(* IEC 61131-3 sources: RL_MAR/experiments/results/ablation/Ablation_random_topo_deepseek-ai_DeepSeek-V3.2_20260603_051006, 94 files *)

(* ---- hard_92.st ---- *)
FUNCTION_BLOCK FB_BreakerControlSystem
VAR_INPUT
    B10_1_Trip : BOOL;
    B10_1_Close : BOOL;
    B10_2_Trip : BOOL;
    B10_2_Close : BOOL;
    B10_12_Trip : BOOL;
    B10_12_Close : BOOL;
    B54_Trip : BOOL;
    B54_Close : BOOL;
    B55_Trip : BOOL;
    B55_Close : BOOL;
    B56_Trip : BOOL;
    B56_Close : BOOL;
    B57_Trip : BOOL;
    B57_Close : BOOL;
END_VAR

VAR_OUTPUT
    Point_1a : INT;
    Point_2a : INT;
    Point_3a : INT;
    Point_4a : INT;
    B10_1_Opened : BOOL;
    B10_1_Closed : BOOL;
    B10_2_Opened : BOOL;
    B10_2_Closed : BOOL;
    B10_12_Opened : BOOL;
    B10_12_Closed : BOOL;
    B54_Opened : BOOL;
    B54_Closed : BOOL;
    B55_Opened : BOOL;
    B55_Closed : BOOL;
    B56_Opened : BOOL;
    B56_Closed : BOOL;
    B57_Opened : BOOL;
    B57_Closed : BOOL;
END_VAR

VAR
    SEL86_OUT : INT;
    MOVE89_OUT : INT;
    SEL66_OUT : INT;
    MOVE69_OUT : INT;
    SEL96_OUT : INT;
    MOVE99_OUT : INT;
    SEL106_OUT : INT;
    MOVE109_OUT : INT;
END_VAR

// Breaker state transitions
IF B10_1_Close THEN
    B10_1_Closed := TRUE;
    B10_1_Opened := FALSE;
ELSIF B10_1_Trip THEN
    B10_1_Closed := FALSE;
    B10_1_Opened := TRUE;
END_IF;

IF B10_2_Close THEN
    B10_2_Closed := TRUE;
    B10_2_Opened := FALSE;
ELSIF B10_2_Trip THEN
    B10_2_Closed := FALSE;
    B10_2_Opened := TRUE;
END_IF;

IF B10_12_Close THEN
    B10_12_Closed := TRUE;
    B10_12_Opened := FALSE;
ELSIF B10_12_Trip THEN
    B10_12_Closed := FALSE;
    B10_12_Opened := TRUE;
END_IF;

IF B54_Close THEN
    B54_Closed := TRUE;
    B54_Opened := FALSE;
ELSIF B54_Trip THEN
    B54_Closed := FALSE;
    B54_Opened := TRUE;
END_IF;

IF B55_Close THEN
    B55_Closed := TRUE;
    B55_Opened := FALSE;
ELSIF B55_Trip THEN
    B55_Closed := FALSE;
    B55_Opened := TRUE;
END_IF;

IF B56_Close THEN
    B56_Closed := TRUE;
    B56_Opened := FALSE;
ELSIF B56_Trip THEN
    B56_Closed := FALSE;
    B56_Opened := TRUE;
END_IF;

IF B57_Close THEN
    B57_Closed := TRUE;
    B57_Opened := FALSE;
ELSIF B57_Trip THEN
    B57_Closed := FALSE;
    B57_Opened := TRUE;
END_IF;

// Point calculations
// Point_1a: B54 closed AND (B10_12 closed AND B10_1 closed) OR B10_2 closed
IF B54_Closed AND ((B10_12_Closed AND B10_1_Closed) OR B10_2_Closed) THEN
    Point_1a := 0;
ELSE
    Point_1a := 138;
END_IF;

// Point_2a: B55 closed AND (B10_12 closed AND B10_1 closed) OR B10_2 closed
IF B55_Closed AND ((B10_12_Closed AND B10_1_Closed) OR B10_2_Closed) THEN
    Point_2a := 0;
ELSE
    Point_2a := 138;
END_IF;

// Point_3a: B56 closed AND (B10_12 closed AND B10_2 closed) OR B10_1 closed
IF B56_Closed AND ((B10_12_Closed AND B10_2_Closed) OR B10_1_Closed) THEN
    Point_3a := 0;
ELSE
    Point_3a := 138;
END_IF;

// Point_4a: B57 closed AND (B10_12 closed AND B10_2 closed) OR B10_1 closed
IF B57_Closed AND ((B10_12_Closed AND B10_2_Closed) OR B10_1_Closed) THEN
    Point_4a := 0;
ELSE
    Point_4a := 138;
END_IF;

END_FUNCTION_BLOCK

(* ---- hard_93.st ---- *)
FUNCTION_BLOCK FB_CircuitControl
VAR_INPUT
    Reset_All_CB : BOOL;
    Current_Fault_on_TRSF1 : INT;
    Current_Fault_on_66BUS1 : INT;
END_VAR

VAR_OUTPUT
    Short_Circuit_TRSF1 : BOOL;
    Short_Circuit_66BUS : BOOL;
    Open_CB1_66KV : BOOL;
    Open_CB2_66KV : BOOL;
    Open_CB_TRSF1 : BOOL;
    Open_CB2_22KV : BOOL;
END_VAR

VAR
    Threshold500 : INT := 500;
    Prev_Open_CB2_22KV : BOOL;
    Prev_Open_CB1_66KV : BOOL;
    Prev_Open_CB_TRSF1 : BOOL;
    Temp_Open_CB2_22KV : BOOL;
    Temp_Open_CB1_66KV : BOOL;
    Temp_Open_CB_TRSF1 : BOOL;
END_VAR

(* a) Implement short circuit detection *)
Short_Circuit_66BUS := (Current_Fault_on_66BUS1 > Threshold500);
Short_Circuit_TRSF1 := (Current_Fault_on_TRSF1 > Threshold500);

(* b) Implement circuit breaker control logic *)

(* First pass: Initial calculations *)
Temp_Open_CB2_22KV := (NOT Reset_All_CB) AND (NOT Prev_Open_CB2_22KV) AND (
    (Open_CB1_66KV AND Open_CB_TRSF1) OR Short_Circuit_66BUS
);

Temp_Open_CB1_66KV := (NOT Reset_All_CB) AND (NOT Temp_Open_CB2_22KV) AND (
    (Prev_Open_CB1_66KV AND Open_CB_TRSF1) OR Short_Circuit_66BUS
);

Temp_Open_CB_TRSF1 := (NOT Reset_All_CB) AND (NOT Temp_Open_CB2_22KV) AND (
    (Temp_Open_CB1_66KV AND Prev_Open_CB_TRSF1) OR Short_Circuit_66BUS
);

Open_CB2_66KV := TRUE;

(* Second pass: Update based on new conditions *)
Temp_Open_CB2_22KV := Temp_Open_CB2_22KV OR (
    (NOT Reset_All_CB) AND (NOT Prev_Open_CB2_22KV) AND (
        (Open_CB2_66KV AND Temp_Open_CB1_66KV AND Temp_Open_CB_TRSF1) OR Short_Circuit_TRSF1
    )
);

Temp_Open_CB1_66KV := Temp_Open_CB1_66KV OR (
    (NOT Reset_All_CB) AND (NOT Temp_Open_CB2_22KV) AND (
        (Open_CB2_66KV AND Prev_Open_CB1_66KV AND Temp_Open_CB_TRSF1) OR Short_Circuit_TRSF1
    )
);

Temp_Open_CB_TRSF1 := Temp_Open_CB_TRSF1 OR (
    (NOT Reset_All_CB) AND (NOT Temp_Open_CB2_22KV) AND (
        (Open_CB2_66KV AND Temp_Open_CB1_66KV AND Prev_Open_CB_TRSF1) OR Short_Circuit_TRSF1
    )
);

(* Assign temporary values to outputs *)
Open_CB2_22KV := Temp_Open_CB2_22KV;
Open_CB1_66KV := Temp_Open_CB1_66KV;
Open_CB_TRSF1 := Temp_Open_CB_TRSF1;

(* Store previous states for next scan *)
Prev_Open_CB2_22KV := Open_CB2_22KV;
Prev_Open_CB1_66KV := Open_CB1_66KV;
Prev_Open_CB_TRSF1 := Open_CB_TRSF1;

(* Failsafe: If Reset_All_CB is TRUE, force all circuit breakers to FALSE *)
IF Reset_All_CB THEN
    Open_CB1_66KV := FALSE;
    Open_CB2_66KV := FALSE;
    Open_CB_TRSF1 := FALSE;
    Open_CB2_22KV := FALSE;
    Prev_Open_CB2_22KV := FALSE;
    Prev_Open_CB1_66KV := FALSE;
    Prev_Open_CB_TRSF1 := FALSE;
END_IF;

END_FUNCTION_BLOCK

(* ---- hard_94.st ---- *)
FUNCTION_BLOCK FB_AdvancedCircuitBreakerControl
VAR_INPUT
    S_AL1_P_B1 : BOOL;
    S_AL1_P_B2 : BOOL;
    S_AL1_MCB : BOOL;
    MCB_BUSY : BOOL;
    MCB_ERROR : BOOL;
    S_AL1_MCBR : BOOL;
    MCBR_BUSY : BOOL;
    MCBR_ERROR : BOOL;
    S_AL1_P_B3 : BOOL;
    S_AL1_MCB2 : BOOL;
    S_AL1_MCBR2 : BOOL;
END_VAR

VAR_OUTPUT
    E_AL1_B1 : BOOL;
    PUWS_AL1_B1_PLUS : BOOL;
    PUWS_AL1_B1_RIGHT : BOOL;
    PAS_AL1_PLUS : BOOL;
    PAS_AL1_TURN : BOOL;
END_VAR

VAR
    PPAL1 : BOOL := 1;
    PP0 : BOOL := 1;
    PP1 : BOOL := 0;
    PP2 : BOOL := 0;
    PP3 : BOOL := 0;
    PP4 : BOOL := 0;
    MCB : BOOL := 1;
    PP5 : BOOL := 0;
    PP7 : BOOL := 0;
    PPL3 : BOOL := 0;
    PPL4 : BOOL := 0;
    MCBR : BOOL := 1;
    PPL5 : BOOL := 0;
    PPL7 : BOOL := 0;
    STABLE : BOOL := 0;
    MCB_CONTROL : BOOL;
END_VAR

STABLE := 0;
WHILE (STABLE = 0) DO
    STABLE := 1;

    IF (PP0 = 1) AND (NOT MCB_CONTROL) AND (NOT PP1) THEN
        PP0 := 0;
        PP1 := 1;
        STABLE := 0;
    END_IF;

    IF (PP1 = 1) AND S_AL1_P_B1 AND (NOT PP2) THEN
        PP1 := 0;
        PP2 := 1;
        STABLE := 0;
    END_IF;

    IF (PP2 = 1) AND S_AL1_P_B2 AND (NOT MCB_CONTROL) AND (NOT PP3) THEN
        PP2 := 0;
        PP3 := 1;
        STABLE := 0;
    END_IF;

    IF (PP2 = 1) AND S_AL1_P_B2 AND MCB_CONTROL AND (NOT PPL3) AND (NOT PP1) THEN
        PP2 := 0;
        PPL3 := 1;
        PP1 := 1;
        STABLE := 0;
    END_IF;

    IF (PP3 = 1) AND S_AL1_MCB AND (NOT PP4) AND (NOT PP1) THEN
        PP3 := 0;
        PP4 := 1;
        PP1 := 1;
        STABLE := 0;
    END_IF;

    IF (PP4 = 1) AND (MCB = 1) AND MCB_BUSY AND (NOT PP5) THEN
        PP4 := 0;
        MCB := 0;
        PP5 := 1;
        STABLE := 0;
    END_IF;

    IF (PP5 = 1) AND S_AL1_MCB2 AND (NOT PP7) AND (NOT MCB) THEN
        PP5 := 0;
        PP7 := 1;
        MCB := 1;
        STABLE := 0;
    END_IF;

    IF (PP7 = 1) AND S_AL1_P_B3 THEN
        PP7 := 0;
        STABLE := 0;
    END_IF;

    IF (PPL3 = 1) AND S_AL1_MCBR AND (NOT PPL4) THEN
        PPL3 := 0;
        PPL4 := 1;
        STABLE := 0;
    END_IF;

    IF (PPL4 = 1) AND (MCBR = 1) AND MCBR_BUSY AND (NOT PPL5) THEN
        PPL4 := 0;
        MCBR := 0;
        PPL5 := 1;
        STABLE := 0;
    END_IF;

    IF (PPL5 = 1) AND S_AL1_MCBR2 AND (NOT PPL7) AND (NOT MCBR) THEN
        PPL5 := 0;
        PPL7 := 1;
        MCBR := 1;
        STABLE := 0;
    END_IF;

    IF (PPL7 = 1) AND S_AL1_P_B3 THEN
        PPL7 := 0;
        STABLE := 0;
    END_IF;
END_WHILE;

IF (PP0 = 1) OR (PP1 = 1) THEN
    E_AL1_B1 := 1;
END_IF;

IF (PP3 = 1) THEN
    MCB_CONTROL := 1;
END_IF;

IF (PPL3 = 1) OR (PPL4 = 1) THEN
    PAS_AL1_PLUS := 1;
    PAS_AL1_TURN := 1;
END_IF;

IF (PPAL1 = 1) OR (PP2 = 1) THEN
    PUWS_AL1_B1_PLUS := 1;
END_IF;

IF (PP2 = 1) OR (PP3 = 1) OR (PPL3 = 1) THEN
    E_AL1_B1 := 0;
END_IF;

IF (PP0 = 1) OR (PP3 = 1) THEN
    MCB_CONTROL := 0;
END_IF;

IF (PP0 = 1) OR (PP3 = 1) OR (PP4 = 1) THEN
    PAS_AL1_PLUS := 0;
    PAS_AL1_TURN := 0;
END_IF;

IF (PPAL1 = 1) OR (PP2 = 1) THEN
    PUWS_AL1_B1_RIGHT := 0;
END_IF;

END_FUNCTION_BLOCK

(* ---- hf_1.st ---- *)
FUNCTION_BLOCK StackMin
VAR_INPUT
    push : BOOL;
    pop : BOOL;
    reset : BOOL;
END_VAR
VAR_OUTPUT
    error : BOOL;
    status : WORD;
END_VAR
VAR_IN_OUT
    item : INT;
    stack : ARRAY[0..3] OF INT;
END_VAR
VAR
    top : INT := -1;
    i : INT;
    minIndex : INT;
    minValue : INT;
    j : INT;
END_VAR

// Reset operation takes highest priority
IF reset THEN
    top := -1;
    error := FALSE;
    status := 16#0000;
ELSIF push THEN
    // Push operation
    IF top >= 3 THEN
        // Stack is full
        error := TRUE;
        status := 16#8A04;
    ELSE
        // Add item to stack
        top := top + 1;
        stack[top] := item;
        error := FALSE;
        status := 16#0000;
    END_IF;
ELSIF pop THEN
    // Pop minimum operation
    IF top < 0 THEN
        // Stack is empty
        error := TRUE;
        status := 16#8A05;
    ELSE
        // Find minimum value and its index
        minIndex := 0;
        minValue := stack[0];

        FOR i := 1 TO top DO
            IF stack[i] < minValue THEN
                minValue := stack[i];
                minIndex := i;
            END_IF;
        END_FOR;

        // Return minimum value via item
        item := minValue;

        // Shift elements down to remove the minimum
        FOR j := minIndex TO top - 1 DO
            stack[j] := stack[j + 1];
        END_FOR;

        // Clear the last position (optional but clean)
        stack[top] := 0;

        // Update top index
        top := top - 1;

        error := FALSE;
        status := 16#0000;
    END_IF;
ELSE
    // No operation requested
    error := FALSE;
    status := 16#0000;
END_IF;
END_FUNCTION_BLOCK

(* ---- hf_10.st ---- *)
FUNCTION_BLOCK FloatingAverage
VAR_INPUT
    cyclicExecution : BOOL;
    trigger : BOOL;
    value : REAL;
    windowSize : INT;
    reset : BOOL;
END_VAR
VAR_OUTPUT
    average : REAL;
    windowSizeReached : BOOL;
    error : BOOL;
    status : WORD;
END_VAR
VAR
    dataBuffer : ARRAY[1..100] OF REAL;
    bufferIndex : INT;
    sum : REAL;
    elementCount : INT;
    prevTrigger : BOOL;
END_VAR

// Initialize variables
bufferIndex := 1;
sum := 0.0;
elementCount := 0;
prevTrigger := FALSE;
average := 0.0;
windowSizeReached := FALSE;
error := FALSE;
status := 16#0000;

// Check for reset condition
IF reset THEN
    bufferIndex := 1;
    sum := 0.0;
    elementCount := 0;
    average := 0.0;
    windowSizeReached := FALSE;
    error := FALSE;
    status := 16#0000;
    RETURN;
END_IF;

// Validate window size
IF (windowSize < 1) OR (windowSize > 100) THEN
    error := TRUE;
    status := 16#8200;
    average := 0.0;
    windowSizeReached := FALSE;
    RETURN;
END_IF;

// Check if we should process new data
IF cyclicExecution OR (trigger AND NOT prevTrigger) THEN
    // Store previous value that will be overwritten
    IF elementCount >= windowSize THEN
        sum := sum - dataBuffer[bufferIndex];
    END_IF;

    // Store new value and update sum
    dataBuffer[bufferIndex] := value;
    sum := sum + value;

    // Update element count
    IF elementCount < windowSize THEN
        elementCount := elementCount + 1;
    END_IF;

    // Update buffer index (circular buffer)
    bufferIndex := bufferIndex + 1;
    IF bufferIndex > windowSize THEN
        bufferIndex := 1;
    END_IF;

    // Calculate average
    IF elementCount > 0 THEN
        average := sum / elementCount;
    ELSE
        average := 0.0;
    END_IF;

    // Check if window size is reached
    windowSizeReached := (elementCount >= windowSize);
END_IF;

// Store current trigger state for edge detection
prevTrigger := trigger;

// Clear error if window size is valid
IF NOT ((windowSize < 1) OR (windowSize > 100)) THEN
    error := FALSE;
    status := 16#0000;
END_IF;

END_FUNCTION_BLOCK

(* ---- hf_11.st ---- *)
FUNCTION_BLOCK FB_BottleProcessing
VAR_INPUT
    bottleSensor : BOOL;
    cleaningConfirmButton : BOOL;
    fillingConfirmButton : BOOL;
    cappingConfirmButton : BOOL;
    packingConfirmButton : BOOL;
    finishedButton : BOOL;
END_VAR

VAR_OUTPUT
    Pump_Motor : BOOL;
    Filling_Valve : BOOL;
    Capping_Machine : BOOL;
    Packing_Machine : BOOL;
    Completion_Light : BOOL;
END_VAR

VAR
    State : INT := 0; (* 0=Waiting, 1=Cleaning, 2=Filling, 3=Capping, 4=Packing, 5=Completed *)
END_VAR

CASE State OF
    0: (* Waiting State *)
        Pump_Motor := FALSE;
        Filling_Valve := FALSE;
        Capping_Machine := FALSE;
        Packing_Machine := FALSE;
        Completion_Light := FALSE;

        IF bottleSensor THEN
            Pump_Motor := TRUE;
            State := 1;
        END_IF;

    1: (* Cleaning State *)
        Pump_Motor := TRUE;
        Filling_Valve := FALSE;
        Capping_Machine := FALSE;
        Packing_Machine := FALSE;
        Completion_Light := FALSE;

        IF cleaningConfirmButton THEN
            Pump_Motor := FALSE;
            Filling_Valve := TRUE;
            State := 2;
        END_IF;

    2: (* Filling State *)
        Pump_Motor := FALSE;
        Filling_Valve := TRUE;
        Capping_Machine := FALSE;
        Packing_Machine := FALSE;
        Completion_Light := FALSE;

        IF fillingConfirmButton THEN
            Filling_Valve := FALSE;
            Capping_Machine := TRUE;
            State := 3;
        END_IF;

    3: (* Capping State *)
        Pump_Motor := FALSE;
        Filling_Valve := FALSE;
        Capping_Machine := TRUE;
        Packing_Machine := FALSE;
        Completion_Light := FALSE;

        IF cappingConfirmButton THEN
            Capping_Machine := FALSE;
            Packing_Machine := TRUE;
            State := 4;
        END_IF;

    4: (* Packing State *)
        Pump_Motor := FALSE;
        Filling_Valve := FALSE;
        Capping_Machine := FALSE;
        Packing_Machine := TRUE;
        Completion_Light := FALSE;

        IF packingConfirmButton THEN
            Packing_Machine := FALSE;
            Completion_Light := TRUE;
            State := 5;
        END_IF;

    5: (* Completed State *)
        Pump_Motor := FALSE;
        Filling_Valve := FALSE;
        Capping_Machine := FALSE;
        Packing_Machine := FALSE;
        Completion_Light := TRUE;

        IF finishedButton THEN
            Completion_Light := FALSE;
            State := 0;
        END_IF;

END_CASE;

END_FUNCTION_BLOCK

(* ---- hf_12.st ---- *)
FUNCTION_BLOCK MaterialMixing
VAR_INPUT
    estop : BOOL; (* Emergency Stop Signal, FALSE: Emergency stop triggered, TRUE: No emergency stop triggered *)
    opeMode : BOOL; (* Operation Mode, FALSE: Manual Operation Mode, TRUE: Automatic Operation Mode *)
    valveAStart : BOOL; (* Valve A Start Button *)
    valveBStart : BOOL; (* Valve B Start Button *)
    valveCStart : BOOL; (* Valve C Start Button *)
    valveDStart : BOOL; (* Valve D Start Button *)
    mixMotorStart : BOOL; (* Mixing Motor Start Button *)
    autoStart : BOOL; (* Automatic Start Button *)
    processMode : BOOL; (* Process Mode *)
    levelSensor : INT; (* Liquid Level Sensor, unit cm *)
    mixMotorComplete : BOOL; (* Mixing Complete Signal *)
END_VAR
VAR_OUTPUT
    valveARun : BOOL; (* Valve A Run Command *)
    valveBRun : BOOL; (* Valve B Run Command *)
    valveCRun : BOOL; (* Valve C Run Command *)
    valveDRun : BOOL; (* Valve D Run Command *)
    mixMotorRun : BOOL; (* Mixing Motor Run Command *)
END_VAR
VAR
    previousValveAStart : BOOL := FALSE;
    previousValveBStart : BOOL := FALSE;
    previousValveCStart : BOOL := FALSE;
    previousValveDStart : BOOL := FALSE;
    previousMixMotorStart : BOOL := FALSE;
    previousAutoStart : BOOL := FALSE;
    autoActive : BOOL := FALSE;
    autoStep : INT := 0;
END_VAR

(* Emergency stop logic - highest priority *)
IF NOT estop THEN
    valveARun := FALSE;
    valveBRun := FALSE;
    valveCRun := FALSE;
    valveDRun := FALSE;
    mixMotorRun := FALSE;
    autoActive := FALSE;
    autoStep := 0;
ELSE
    (* Manual mode *)
    IF NOT opeMode THEN
        (* Valve A toggle control *)
        IF valveAStart AND NOT previousValveAStart THEN
            valveARun := NOT valveARun;
        END_IF;
        previousValveAStart := valveAStart;

        (* Valve B toggle control *)
        IF valveBStart AND NOT previousValveBStart THEN
            valveBRun := NOT valveBRun;
        END_IF;
        previousValveBStart := valveBStart;

        (* Valve C toggle control *)
        IF valveCStart AND NOT previousValveCStart THEN
            valveCRun := NOT valveCRun;
        END_IF;
        previousValveCStart := valveCStart;

        (* Valve D toggle control *)
        IF valveDStart AND NOT previousValveDStart THEN
            valveDRun := NOT valveDRun;
        END_IF;
        previousValveDStart := valveDStart;

        (* Mixing motor toggle control *)
        IF mixMotorStart AND NOT previousMixMotorStart THEN
            mixMotorRun := NOT mixMotorRun;
        END_IF;
        previousMixMotorStart := mixMotorStart;

        (* Reset automatic mode variables in manual mode *)
        autoActive := FALSE;
        autoStep := 0;

    (* Automatic mode *)
    ELSE
        (* Auto start button handling - toggle functionality *)
        IF autoStart AND NOT previousAutoStart THEN
            autoActive := NOT autoActive;
            IF autoActive THEN
                autoStep := 1;
            ELSE
                autoStep := 0;
            END_IF;
        END_IF;
        previousAutoStart := autoStart;

        (* Automatic process sequence *)
        IF autoActive THEN
            CASE autoStep OF
                1: (* Step 1: Open valve A *)
                    valveARun := TRUE;
                    valveBRun := FALSE;
                    valveCRun := FALSE;
                    valveDRun := FALSE;
                    mixMotorRun := FALSE;

                    IF levelSensor >= 50 THEN
                        valveARun := FALSE;
                        autoStep := 2;
                    END_IF;

                2: (* Step 2: Open valve B *)
                    valveBRun := TRUE;

                    IF levelSensor >= 80 THEN
                        valveBRun := FALSE;
                        autoStep := 3;
                    END_IF;

                3: (* Step 3: Process mode decision *)
                    IF NOT processMode THEN
                        (* Process mode false: Start mixing motor *)
                        mixMotorRun := TRUE;

                        IF mixMotorComplete THEN
                            mixMotorRun := FALSE;
                            autoStep := 4;
                        END_IF;
                    ELSE
                        (* Process mode true: Open valve C *)
                        valveCRun := TRUE;

                        IF levelSensor >= 100 THEN
                            valveCRun := FALSE;
                            autoStep := 4;
                        END_IF;
                    END_IF;

                4: (* Step 4: Handle mixing for process mode true *)
                    IF processMode THEN
                        mixMotorRun := TRUE;

                        IF mixMotorComplete THEN
                            mixMotorRun := FALSE;
                            autoStep := 5;
                        END_IF;
                    ELSE
                        autoStep := 5;
                    END_IF;

                5: (* Step 5: Open valve D and end process *)
                    valveDRun := TRUE;
                    autoActive := FALSE;
                    autoStep := 0;

            END_CASE;
        ELSE
            (* Auto not active - ensure all outputs are off *)
            valveARun := FALSE;
            valveBRun := FALSE;
            valveCRun := FALSE;
            valveDRun := FALSE;
            mixMotorRun := FALSE;
        END_IF;
    END_IF;
END_IF;

END_FUNCTION_BLOCK

(* ---- hf_13.st ---- *)
FUNCTION_BLOCK TON
VAR_INPUT
    IN : BOOL;
    PT : DINT;
    CYCLE_TIME : DINT;
END_VAR
VAR_OUTPUT
    Q : BOOL;
    ET : DINT;
END_VAR
VAR
    elapsedTimeInternal : DINT := 0;
    IN_PREV : BOOL := FALSE;
END_VAR

IF IN THEN
    IF NOT IN_PREV THEN
        elapsedTimeInternal := 0;
    END_IF;

    IF elapsedTimeInternal < PT THEN
        elapsedTimeInternal := elapsedTimeInternal + CYCLE_TIME;
        Q := FALSE;
    ELSE
        elapsedTimeInternal := PT;
        Q := TRUE;
    END_IF;

    ET := elapsedTimeInternal;
ELSE
    Q := FALSE;
    ET := 0;
    elapsedTimeInternal := 0;
END_IF;

IN_PREV := IN;
END_FUNCTION_BLOCK

FUNCTION_BLOCK LightsControl
VAR_INPUT
    button1 : BOOL; (* Button 1: Automatic/Manual Mode Select *)
    button2 : BOOL; (* Button 2: Manual Control/Green Light Req *)
    button3 : BOOL; (* Button 3: Manual Control/Red Light Req *)
    CYCLE_TIME : DINT; (* Time elapsed in current cycle (in ms) *)
END_VAR
VAR_OUTPUT
    greenLight : BOOL; (* Green light *)
    redLight : BOOL; (* Red light *)
    yellowLight : BOOL; (* Yellow light *)
END_VAR
VAR
    (* Timers for control *)
    timerAuto : TON;
    timerGreen : TON;
    timerRed : TON;
    timerYellow : TON;

    currentState : INT := 0;
    autoRunTimer : BOOL := TRUE;

    (* Internal variables for blinking control *)
    blinkToggleRed : BOOL := FALSE;
    blinkToggleYellow : BOOL := FALSE;
    blinkToggleGreen : BOOL := FALSE;
    prevTimerRedQ : BOOL := FALSE;
    prevTimerYellowQ : BOOL := FALSE;
    prevTimerGreenQ : BOOL := FALSE;
END_VAR

(* Reset all outputs initially *)
greenLight := FALSE;
redLight := FALSE;
yellowLight := FALSE;

IF button1 THEN (* Automatic Mode *)
    (* Reset manual mode timers *)
    timerGreen(IN := FALSE, PT := 0, CYCLE_TIME := CYCLE_TIME);
    timerRed(IN := FALSE, PT := 0, CYCLE_TIME := CYCLE_TIME);
    timerYellow(IN := FALSE, PT := 0, CYCLE_TIME := CYCLE_TIME);

    (* Reset blinking toggle variables *)
    blinkToggleRed := FALSE;
    blinkToggleYellow := FALSE;
    blinkToggleGreen := FALSE;

    (* Automatic mode state machine *)
    timerAuto(IN := autoRunTimer, PT := 1000, CYCLE_TIME := CYCLE_TIME);

    CASE currentState OF
        0: (* State 0: Green light ON for 1 second *)
            greenLight := TRUE;
            redLight := FALSE;
            yellowLight := FALSE;

            IF timerAuto.Q THEN
                currentState := 1;
                timerAuto(IN := FALSE, PT := 1000, CYCLE_TIME := CYCLE_TIME);
            END_IF;

        1: (* State 1: Red light ON for 1 second *)
            greenLight := FALSE;
            redLight := TRUE;
            yellowLight := FALSE;

            IF timerAuto.Q THEN
                currentState := 2;
                timerAuto(IN := FALSE, PT := 1000, CYCLE_TIME := CYCLE_TIME);
            END_IF;

        2: (* State 2: Yellow light ON for 1 second *)
            greenLight := FALSE;
            redLight := FALSE;
            yellowLight := TRUE;

            IF timerAuto.Q THEN
                currentState := 0;
                timerAuto(IN := FALSE, PT := 1000, CYCLE_TIME := CYCLE_TIME);
            END_IF;
    END_CASE;

    (* Restart timer for next cycle *)
    IF NOT timerAuto.IN THEN
        timerAuto(IN := TRUE, PT := 1000, CYCLE_TIME := CYCLE_TIME);
    END_IF;

ELSE (* Manual Mode *)
    (* Reset automatic mode timer *)
    timerAuto(IN := FALSE, PT := 0, CYCLE_TIME := CYCLE_TIME);

    (* Reset automatic mode state *)
    currentState := 0;

    (* Manual mode logic based on button combinations *)
    IF NOT button2 AND NOT button3 THEN
        (* Both FALSE: All lights off *)
        greenLight := FALSE;
        redLight := FALSE;
        yellowLight := FALSE;

        (* Reset all timers and blinking states *)
        timerGreen(IN := FALSE, PT := 0, CYCLE_TIME := CYCLE_TIME);
        timerRed(IN := FALSE, PT := 0, CYCLE_TIME := CYCLE_TIME);
        timerYellow(IN := FALSE, PT := 0, CYCLE_TIME := CYCLE_TIME);
        blinkToggleRed := FALSE;
        blinkToggleYellow := FALSE;
        blinkToggleGreen := FALSE;

    ELSIF button2 AND NOT button3 THEN
        (* button2 TRUE, button3 FALSE: Green light ON, Red light blinking at 0.5Hz *)
        greenLight := TRUE;
        yellowLight := FALSE;

        (* Red light blinking logic *)
        timerRed(IN := TRUE, PT := 2000, CYCLE_TIME := CYCLE_TIME);

        (* Detect rising edge of timer output to toggle blink *)
        IF timerRed.Q AND NOT prevTimerRedQ THEN
            blinkToggleRed := NOT blinkToggleRed;
        END_IF;
        prevTimerRedQ := timerRed.Q;

        (* Red light blinks at 0.5Hz using timer Q directly *)
        redLight := blinkToggleRed;

        (* Reset other timers *)
        timerGreen(IN := FALSE, PT := 0, CYCLE_TIME := CYCLE_TIME);
        timerYellow(IN := FALSE, PT := 0, CYCLE_TIME := CYCLE_TIME);
        blinkToggleYellow := FALSE;
        blinkToggleGreen := FALSE;

    ELSIF NOT button2 AND button3 THEN
        (* button2 FALSE, button3 TRUE: Red light ON, Yellow light blinking at 1Hz *)
        redLight := TRUE;
        greenLight := FALSE;

        (* Yellow light blinking logic *)
        timerYellow(IN := TRUE, PT := 1000, CYCLE_TIME := CYCLE_TIME);

        (* Detect rising edge of timer output to toggle blink *)
        IF timerYellow.Q AND NOT prevTimerYellowQ THEN
            blinkToggleYellow := NOT blinkToggleYellow;
        END_IF;
        prevTimerYellowQ := timerYellow.Q;

        (* Yellow light blinks at 1Hz using NOT timer Q *)
        yellowLight := blinkToggleYellow;

        (* Reset other timers *)
        timerGreen(IN := FALSE, PT := 0, CYCLE_TIME := CYCLE_TIME);
        timerRed(IN := FALSE, PT := 0, CYCLE_TIME := CYCLE_TIME);
        blinkToggleRed := FALSE;
        blinkToggleGreen := FALSE;

    ELSIF button2 AND button3 THEN
        (* Both TRUE: Yellow light ON, Green light blinking at 1Hz *)
        yellowLight := TRUE;
        redLight := FALSE;

        (* Green light blinking logic *)
        timerGreen(IN := TRUE, PT := 1000, CYCLE_TIME := CYCLE_TIME);

        (* Detect rising edge of timer output to toggle blink *)
        IF timerGreen.Q AND NOT prevTimerGreenQ THEN
            blinkToggleGreen := NOT blinkToggleGreen;
        END_IF;
        prevTimerGreenQ := timerGreen.Q;

        (* Green light blinks at 1Hz using NOT timer Q *)
        greenLight := blinkToggleGreen;

        (* Reset other timers *)
        timerRed(IN := FALSE, PT := 0, CYCLE_TIME := CYCLE_TIME);
        timerYellow(IN := FALSE, PT := 0, CYCLE_TIME := CYCLE_TIME);
        blinkToggleRed := FALSE;
        blinkToggleYellow := FALSE;
    END_IF;
END_IF;
END_FUNCTION_BLOCK

(* ---- hf_14.st ---- *)
FUNCTION_BLOCK TruckGarage
VAR_INPUT
    enter_flag : BOOL;
    exit_flag : BOOL;
    VehicleNumber_in : INT;
END_VAR
VAR_OUTPUT
    truck_row : INT;
    truck_col : INT;
    truck_VehicleNumber : INT;
END_VAR
VAR_IN_OUT
    garage : ARRAY[1..3, 1..5] OF STRUCT
        Occupied : BOOL;
        VehicleNumber : INT;
    END_STRUCT;
END_VAR
VAR
    i : INT;
    j : INT;
    space_found : BOOL;
    exit_found : BOOL;
END_VAR

// Initialize output variables
truck_row := 0;
truck_col := 0;
truck_VehicleNumber := 0;

// Entry logic
IF enter_flag THEN
    space_found := FALSE;

    // Search from last row to first row
    FOR i := 3 TO 1 BY -1 DO
        // Search from last column to first column
        FOR j := 5 TO 1 BY -1 DO
            IF NOT garage[i, j].Occupied THEN
                // Found empty space
                garage[i, j].Occupied := TRUE;
                garage[i, j].VehicleNumber := VehicleNumber_in;
                space_found := TRUE;
                EXIT;
            END_IF;
        END_FOR;

        IF space_found THEN
            EXIT;
        END_IF;
    END_FOR;
END_IF;

// Exit logic
IF exit_flag THEN
    exit_found := FALSE;

    // Search from first row to last row
    FOR i := 1 TO 3 DO
        // Search from first column to last column
        FOR j := 1 TO 5 DO
            IF garage[i, j].Occupied AND garage[i, j].VehicleNumber = VehicleNumber_in THEN
                // Found vehicle to exit
                truck_row := i;
                truck_col := j;
                truck_VehicleNumber := garage[i, j].VehicleNumber;

                // Clear the parking space
                garage[i, j].Occupied := FALSE;
                garage[i, j].VehicleNumber := 0;

                exit_found := TRUE;
                EXIT;
            END_IF;
        END_FOR;

        IF exit_found THEN
            EXIT;
        END_IF;
    END_FOR;
END_IF;
END_FUNCTION_BLOCK

(* ---- hf_15.st ---- *)
FUNCTION_BLOCK FB_MergeBytes
VAR_INPUT
    byteArray : ARRAY[1..20] OF DINT; (* Byte array to be merged *)
END_VAR
VAR_OUTPUT
    dwordArray : ARRAY[1..10] OF DINT; (* Merged double word array *)
    mergeDwordNum : DINT; (* Actual number of merged double words *)
END_VAR
VAR
    i, j, k : DINT; (* Changed from INT to DINT to match array indices *)
    tempDword : DINT;
    currentByteValue : DINT;
END_VAR
VAR CONSTANT
    BYTE_ARRAY_SIZE : DINT := 20; (* Size of the input byte array *)
    DWORD_ARRAY_SIZE : DINT := 10; (* Size of the output DINT array *)
END_VAR

(* Main logic for merging bytes into double words *)
mergeDwordNum := 0;
tempDword := 0;

(* Calculate maximum possible double words from byte array *)
IF BYTE_ARRAY_SIZE >= 4 THEN
    FOR i := 1 TO BYTE_ARRAY_SIZE DO
        (* Extract current byte value (mask to keep only lowest 8 bits) *)
        currentByteValue := byteArray[i] AND 16#FF;

        (* Position byte within double word *)
        CASE (i MOD 4) OF
            1: (* First byte - least significant *)
                tempDword := currentByteValue;

            2: (* Second byte *)
                tempDword := tempDword OR (currentByteValue SHL 8);

            3: (* Third byte *)
                tempDword := tempDword OR (currentByteValue SHL 16);

            0: (* Fourth byte - most significant *)
                tempDword := tempDword OR (currentByteValue SHL 24);

                (* Store completed double word if space available *)
                IF mergeDwordNum < DWORD_ARRAY_SIZE THEN
                    mergeDwordNum := mergeDwordNum + 1;
                    dwordArray[mergeDwordNum] := tempDword;
                END_IF;

                tempDword := 0; (* Reset for next double word *)
        END_CASE;
    END_FOR;
END_IF;

(* Clear remaining positions in dwordArray if any *)
FOR k := (mergeDwordNum + 1) TO DWORD_ARRAY_SIZE DO
    dwordArray[k] := 0;
END_FOR;

END_FUNCTION_BLOCK

(* ---- hf_16.st ---- *)
FUNCTION_BLOCK FB_LinearizeValue
VAR_INPUT
    InputValue : REAL; // Floating point input, raw measurement value
END_VAR

VAR_OUTPUT
    LinearizedValue : REAL; // Converted linear value
    Error : BOOL; // Error status indicator
    Status : WORD; // Status code
END_VAR

VAR
    // Internal constants for readability and maintainability
    InputMin : REAL := 1200.0;
    InputMax : REAL := 7000.0;
    OutputMin : REAL := 150.0;
    OutputMax : REAL := 720.0;

    // Pre-calculated slopes for each segment for efficiency
    Slope1 : REAL := (240.0 - 150.0) / (3600.0 - 1200.0); // 90/2400
    Slope2 : REAL := (560.0 - 240.0) / (4800.0 - 3600.0); // 320/1200
    Slope3 : REAL := (720.0 - 560.0) / (7000.0 - 4800.0); // 160/2200
END_VAR

// Main execution logic
IF InputValue < InputMin THEN
    // Below minimum range
    LinearizedValue := OutputMin;
    Error := TRUE;
    Status := 16#8001;
ELSIF InputValue > InputMax THEN
    // Above maximum range
    LinearizedValue := OutputMax;
    Error := TRUE;
    Status := 16#8001;
ELSE
    // Input is within valid range
    Error := FALSE;
    Status := 16#0000;

    // Determine which segment the input falls into
    IF InputValue <= 3600.0 THEN
        // Range 1: 1200 to 3600
        LinearizedValue := 150.0 + (InputValue - 1200.0) * Slope1;
    ELSIF InputValue <= 4800.0 THEN
        // Range 2: 3600 to 4800
        LinearizedValue := 240.0 + (InputValue - 3600.0) * Slope2;
    ELSE
        // Range 3: 4800 to 7000
        LinearizedValue := 560.0 + (InputValue - 4800.0) * Slope3;
    END_IF;
END_IF;

END_FUNCTION_BLOCK

(* ---- hf_17.st ---- *)
FUNCTION_BLOCK FB_WarehouseManagement
VAR_INPUT
    requestIn : BOOL := FALSE;
    requestOut : BOOL := FALSE;
END_VAR

VAR_OUTPUT
    productNum : INT := 0;
    libFreeNum : INT := 9;
    error : BOOL := FALSE;
    status : WORD := 16#0000;
END_VAR

VAR_IN_OUT
    library : ARRAY[1..9] OF BOOL;
END_VAR

VAR
    i : INT;
    found : BOOL;
    errFull : WORD := 16#8001;
    errEmpty : WORD := 16#8002;
    initDone : BOOL := FALSE;
END_VAR

// Reset error status at start of each cycle
error := FALSE;
status := 16#0000;

// Initialize library array on first execution
IF NOT initDone THEN
    i := 1;
    WHILE i <= 9 DO
        library[i] := FALSE;
        i := i + 1;
    END_WHILE;
    initDone := TRUE;
END_IF;

// Handle product storage request
IF requestIn AND NOT requestOut THEN
    // Check if storage is full
    IF productNum >= 9 THEN
        error := TRUE;
        status := errFull;
    ELSE
        // Search for free position from highest to lowest index (First-In-Last-Out)
        found := FALSE;
        i := 9;
        WHILE i >= 1 AND NOT found DO
            IF NOT library[i] THEN
                library[i] := TRUE;
                productNum := productNum + 1;
                libFreeNum := libFreeNum - 1;
                found := TRUE;
            END_IF;
            i := i - 1;
        END_WHILE;

        // If no free position found (should not happen with proper checks)
        IF NOT found THEN
            error := TRUE;
            status := errFull;
        END_IF;
    END_IF;
END_IF;

// Handle product retrieval request
IF requestOut AND NOT requestIn THEN
    // Check if storage is empty
    IF productNum <= 0 THEN
        error := TRUE;
        status := errEmpty;
    ELSE
        // Search for occupied position from lowest to highest index (First-In-First-Out)
        found := FALSE;
        i := 1;
        WHILE i <= 9 AND NOT found DO
            IF library[i] THEN
                library[i] := FALSE;
                productNum := productNum - 1;
                libFreeNum := libFreeNum + 1;
                found := TRUE;
            END_IF;
            i := i + 1;
        END_WHILE;

        // If no occupied position found (should not happen with proper checks)
        IF NOT found THEN
            error := TRUE;
            status := errEmpty;
        END_IF;
    END_IF;
END_IF;

// Handle concurrent requests (both true) - prioritize storage
IF requestIn AND requestOut THEN
    // Check if storage is full for storage operation
    IF productNum >= 9 THEN
        error := TRUE;
        status := errFull;
    ELSE
        // Perform storage operation (same logic as above)
        found := FALSE;
        i := 9;
        WHILE i >= 1 AND NOT found DO
            IF NOT library[i] THEN
                library[i] := TRUE;
                productNum := productNum + 1;
                libFreeNum := libFreeNum - 1;
                found := TRUE;
            END_IF;
            i := i - 1;
        END_WHILE;

        IF NOT found THEN
            error := TRUE;
            status := errFull;
        END_IF;
    END_IF;
END_IF;

END_FUNCTION_BLOCK

(* ---- hf_18.st ---- *)
FUNCTION_BLOCK FB_ColorLightControl
VAR_INPUT
    controlButton : BOOL; // Push button for sequence control
END_VAR

VAR_OUTPUT
    greenLight : BOOL; // Green light control signal
    redLight : BOOL; // Red light control signal
    yellowLight : BOOL; // Yellow light control signal
END_VAR

VAR
    state : INT := 1; // State machine control variable
    lastControlButton : BOOL := FALSE; // Previous button state for edge detection
END_VAR

// Main logic
IF (controlButton = TRUE) AND (lastControlButton = FALSE) THEN
    // Rising edge detected - execute state transition
    CASE state OF
        1: // State 1: Green Only -> Transition to State 2
            greenLight := FALSE;
            redLight := TRUE;
            yellowLight := FALSE;
            state := 2;

        2: // State 2: Red Only -> Transition to State 3
            greenLight := FALSE;
            redLight := FALSE;
            yellowLight := TRUE;
            state := 3;

        3: // State 3: Yellow Only -> Transition to State 4
            greenLight := TRUE;
            redLight := TRUE;
            yellowLight := TRUE;
            state := 4;

        4: // State 4: All Lights On -> Transition to State 5
            greenLight := FALSE;
            redLight := FALSE;
            yellowLight := FALSE;
            state := 5;

        5: // State 5: All Lights Off -> Transition to State 1
            greenLight := TRUE;
            redLight := FALSE;
            yellowLight := FALSE;
            state := 1;
    END_CASE;
ELSE
    // No rising edge - maintain current state outputs
    CASE state OF
        1: // State 1: Green Only
            greenLight := TRUE;
            redLight := FALSE;
            yellowLight := FALSE;

        2: // State 2: Red Only
            greenLight := FALSE;
            redLight := TRUE;
            yellowLight := FALSE;

        3: // State 3: Yellow Only
            greenLight := FALSE;
            redLight := FALSE;
            yellowLight := TRUE;

        4: // State 4: All Lights On
            greenLight := TRUE;
            redLight := TRUE;
            yellowLight := TRUE;

        5: // State 5: All Lights Off
            greenLight := FALSE;
            redLight := FALSE;
            yellowLight := FALSE;
    END_CASE;
END_IF;

// Update lastControlButton for next cycle's edge detection
lastControlButton := controlButton;

END_FUNCTION_BLOCK

(* ---- hf_19.st ---- *)
FUNCTION_BLOCK FB_DatabaseManager
VAR_INPUT
    dataInput : ARRAY[0..5] OF BYTE;
    storeTrigger : BOOL;
    resetTrigger : BOOL;
END_VAR
VAR_OUTPUT
    usedSpace : INT := 0;
    remainingSpace : INT := 20;
    error : BOOL;
    status : WORD;
END_VAR
VAR_IN_OUT
    dataBase : ARRAY[1..20] OF BYTE;
END_VAR
VAR
    i : INT;
    dataLength : INT;
END_VAR

IF resetTrigger THEN
    (* Reset Operation *)
    FOR i := 1 TO 20 DO
        dataBase[i] := 0;
    END_FOR;
    usedSpace := 0;
    remainingSpace := 20;
    error := FALSE;
    status := 0;
ELSIF storeTrigger THEN
    (* Data Storage Operation *)
    dataLength := dataInput[0];

    (* Length Validation *)
    IF (dataLength <= 0) OR (dataLength > 5) THEN
        error := TRUE;
        status := 16#8001;
    ELSE
        (* Space Verification *)
        IF (usedSpace + dataLength) > 20 THEN
            error := TRUE;
            status := 16#8002;
        ELSE
            (* Data Storage *)
            FOR i := 1 TO dataLength DO
                dataBase[usedSpace + i] := dataInput[i];
            END_FOR;

            (* Update counters *)
            usedSpace := usedSpace + dataLength;
            remainingSpace := 20 - usedSpace;
            error := FALSE;
            status := 0;
        END_IF;
    END_IF;
END_IF;

END_FUNCTION_BLOCK

(* ---- hf_2.st ---- *)
FUNCTION_BLOCK FindMinMaxValues
VAR_INPUT
    values : ARRAY[1..10] OF DINT;
END_VAR
VAR_OUTPUT
    minValue : DINT;
    minValueIndex : DINT;
    maxValue : DINT;
    maxValueIndex : DINT;
END_VAR
VAR
    i : INT;
END_VAR

// Initialize with first element
minValue := values[1];
maxValue := values[1];
minValueIndex := 1;
maxValueIndex := 1;

// Iterate through remaining elements
FOR i := 2 TO 10 DO
    // Check for new minimum
    IF values[i] < minValue THEN
        minValue := values[i];
        minValueIndex := i;
    END_IF;

    // Check for new maximum
    IF values[i] > maxValue THEN
        maxValue := values[i];
        maxValueIndex := i;
    END_IF;
END_FOR;

END_FUNCTION_BLOCK

(* ---- hf_20.st ---- *)
FUNCTION_BLOCK FB_ProductionLineControl
VAR_INPUT
    Mode : BOOL;           // Manual/Auto mode selection
    ForwardButton : BOOL;  // Forward rotation button
    ReverseButton : BOOL;  // Reverse rotation button
    SensorA : BOOL;        // Sensor A input
    SensorB : BOOL;        // Sensor B input
    SensorC : BOOL;        // Sensor C input
    ButtonA : BOOL;        // Button A input
    ButtonB : BOOL;        // Button B input
    ButtonC : BOOL;        // Button C input
END_VAR

VAR_OUTPUT
    MotorForward : BOOL;   // Motor forward output
    MotorReverse : BOOL;   // Motor reverse output
    CompletionLight : BOOL; // Process completion indicator
END_VAR

VAR
    State : INT;           // State machine current state
END_VAR

// Main logic
IF State = 0 THEN
    // Initialization state
    MotorForward := FALSE;
    MotorReverse := FALSE;
    CompletionLight := FALSE;
    State := 1;
ELSE
    IF NOT Mode THEN
        // Manual mode operation
        IF ForwardButton AND NOT ReverseButton THEN
            // Forward motion
            MotorForward := TRUE;
            MotorReverse := FALSE;
        ELSIF ReverseButton AND NOT ForwardButton THEN
            // Reverse motion
            MotorForward := FALSE;
            MotorReverse := TRUE;
        ELSE
            // Stop condition (both buttons or neither)
            MotorForward := FALSE;
            MotorReverse := FALSE;
        END_IF;

        // Manual mode doesn't use CompletionLight
        CompletionLight := FALSE;
    ELSE
        // Automatic mode operation
        CASE State OF
            1: // Waiting at Station A
                MotorForward := FALSE;
                MotorReverse := FALSE;
                CompletionLight := FALSE;

                IF SensorA THEN
                    State := 2;
                END_IF;

            2: // Processing at Station A
                MotorForward := FALSE;
                MotorReverse := FALSE;

                IF ButtonA THEN
                    MotorForward := TRUE;
                    MotorReverse := FALSE;
                    State := 3;
                END_IF;

            3: // Moving to Station B
                // MotorForward remains TRUE from State 2
                MotorReverse := FALSE;

                IF SensorB THEN
                    MotorForward := FALSE;
                    State := 4;
                END_IF;

            4: // Processing at Station B
                MotorForward := FALSE;
                MotorReverse := FALSE;

                IF ButtonB THEN
                    MotorForward := TRUE;
                    MotorReverse := FALSE;
                    State := 5;
                END_IF;

            5: // Moving to Station C
                // MotorForward remains TRUE from State 4
                MotorReverse := FALSE;

                IF SensorC THEN
                    MotorForward := FALSE;
                    State := 6;
                END_IF;

            6: // Processing at Station C
                MotorForward := FALSE;
                MotorReverse := FALSE;

                IF ButtonC THEN
                    CompletionLight := TRUE;
                    State := 7;
                END_IF;

            7: // Cycle Completion
                MotorForward := FALSE;
                MotorReverse := FALSE;

                IF NOT SensorC THEN
                    CompletionLight := FALSE;
                    State := 1;
                END_IF;

        END_CASE;
    END_IF;
END_IF;

END_FUNCTION_BLOCK

(* ---- hf_21.st ---- *)
FUNCTION_BLOCK FB_SplitNumber
VAR_INPUT
    InputNumber : INT;
END_VAR

VAR_OUTPUT
    Thousands : INT;
    Hundreds : INT;
    Tens : INT;
    Ones : INT;
    Min : INT;
    error : BOOL;
    status : WORD;
END_VAR

VAR
    tempNumber : INT;
    minValue : INT;
    digit1 : INT;
    digit2 : INT;
    digit3 : INT;
    digit4 : INT;
END_VAR

// Input validation
IF (InputNumber < 0) OR (InputNumber > 9999) THEN
    // Error condition
    error := TRUE;
    status := 16#8001;
    Thousands := 0;
    Hundreds := 0;
    Tens := 0;
    Ones := 0;
    Min := 0;
ELSE
    // Valid input
    error := FALSE;
    status := 0;

    // Digit separation
    Thousands := InputNumber / 1000;
    tempNumber := InputNumber MOD 1000;
    Hundreds := tempNumber / 100;
    tempNumber := tempNumber MOD 100;
    Tens := tempNumber / 10;
    Ones := tempNumber MOD 10;

    // Minimum non-zero digit detection
    minValue := 32767; // Maximum INT value

    // Check Thousands digit
    IF Thousands > 0 THEN
        minValue := minimal(minValue, Thousands);
    END_IF;

    // Check Hundreds digit
    IF Hundreds > 0 THEN
        minValue := minimal(minValue, Hundreds);
    END_IF;

    // Check Tens digit
    IF Tens > 0 THEN
        minValue := minimal(minValue, Tens);
    END_IF;

    // Check Ones digit
    IF Ones > 0 THEN
        minValue := minimal(minValue, Ones);
    END_IF;

    // Set Min output
    IF minValue = 32767 THEN
        // All digits are zero
        Min := 0;
    ELSE
        Min := minValue;
    END_IF;
END_IF;
END_FUNCTION_BLOCK

FUNCTION minimal : INT
VAR_INPUT
    IN1 : INT;
    IN2 : INT;
END_VAR

IF IN1 <= IN2 THEN
    minimal := IN1;
ELSE
    minimal := IN2;
END_IF;
END_FUNCTION

(* ---- hf_3.st ---- *)
FUNCTION_BLOCK MultiPumpCtrl
VAR_INPUT
    mode : BOOL;
    start : BOOL;
    stop : BOOL;
    priorities : ARRAY[1..5] OF INT;
    selections : ARRAY[1..5] OF BOOL;
END_VAR
VAR_OUTPUT
    RunComds : ARRAY[1..5] OF BOOL;
END_VAR
VAR
    i : INT;
    j : INT;
    maxPriority : INT;
    maxIndex : INT;
    runCount : INT;
    usedInAuto : ARRAY[1..5] OF BOOL;
END_VAR

// Main logic
IF stop THEN
    // Stop has highest priority: stop all pumps
    FOR i := 1 TO 5 DO
        RunComds[i] := FALSE;
    END_FOR;
ELSIF start THEN
    IF NOT mode THEN
        // Manual mode: set run commands based on manual selections
        FOR i := 1 TO 5 DO
            RunComds[i] := selections[i];
        END_FOR;
    ELSE
        // Automatic mode: find and run 3 pumps with highest priorities
        // Initialize arrays
        FOR i := 1 TO 5 DO
            usedInAuto[i] := FALSE;
            RunComds[i] := FALSE;
        END_FOR;

        // Find 3 highest priority pumps
        runCount := 0;
        WHILE runCount < 3 DO
            maxPriority := -32768; // Minimum INT value
            maxIndex := 0;

            // Find highest priority pump not already selected
            FOR i := 1 TO 5 DO
                IF (priorities[i] > maxPriority) AND NOT usedInAuto[i] THEN
                    maxPriority := priorities[i];
                    maxIndex := i;
                END_IF;
            END_FOR;

            // Activate the found pump
            IF maxIndex > 0 THEN
                RunComds[maxIndex] := TRUE;
                usedInAuto[maxIndex] := TRUE;
                runCount := runCount + 1;
            ELSE
                // No more pumps available (should not happen with 5 pumps)
                EXIT;
            END_IF;
        END_WHILE;
    END_IF;
ELSE
    // When start is FALSE, maintain current state
    // No action needed - RunComds retain their previous values
END_IF;

END_FUNCTION_BLOCK

(* ---- hf_4.st ---- *)
FUNCTION_BLOCK FB_CalculateDayOfYear
VAR_INPUT
    Year : INT;
    Month : INT;
    Day : INT;
END_VAR
VAR_OUTPUT
    DayOfYear : INT;
    error : BOOL;
    status : WORD;
END_VAR
VAR_TEMP
    i : INT;
    isLeapYear : BOOL;
    maxDay : INT;
END_VAR
VAR
    DaysInMonth : ARRAY[1..12] OF INT := [31, 28, 31, 30, 31, 30, 31, 31, 30, 31, 30, 31];
END_VAR

(* Initialize outputs *)
DayOfYear := 0;
error := FALSE;
status := 0;

(* 1. Month validation (highest priority) *)
IF (Month < 1) OR (Month > 12) THEN
    error := TRUE;
    status := 16#8002;  (* Invalid month *)
    RETURN;
END_IF;

(* 2. Day validation (second priority) *)
(* First check if day is positive *)
IF Day <= 0 THEN
    error := TRUE;
    status := 16#8003;  (* Invalid day *)
    RETURN;
END_IF;

(* Determine leap year status *)
isLeapYear := ((Year MOD 4 = 0) AND (Year MOD 100 <> 0)) OR (Year MOD 400 = 0);

(* Get maximum days for the month *)
maxDay := DaysInMonth[Month];
IF (Month = 2) AND isLeapYear THEN
    maxDay := 29;
END_IF;

(* Check if day exceeds maximum for the month *)
IF Day > maxDay THEN
    error := TRUE;
    status := 16#8003;  (* Invalid day *)
    RETURN;
END_IF;

(* 3. Year validation (lowest priority) *)
IF (Year < 1000) OR (Year > 3000) THEN
    error := TRUE;
    status := 16#8001;  (* Invalid year *)
    RETURN;
END_IF;

(* All inputs valid - calculate day of year *)
FOR i := 1 TO (Month - 1) DO
    DayOfYear := DayOfYear + DaysInMonth[i];
END_FOR;

DayOfYear := DayOfYear + Day;

(* Add extra day for leap years if month is after February *)
IF isLeapYear AND (Month > 2) THEN
    DayOfYear := DayOfYear + 1;
END_IF;

END_FUNCTION_BLOCK

(* ---- hf_5.st ---- *)
FUNCTION_BLOCK SelectSort
VAR_INPUT
    exe : BOOL;
    seq : ARRAY[1..100] OF INT;
END_VAR
VAR_OUTPUT
    error : BOOL;
    status : WORD;
END_VAR
VAR
    i : INT;
    j : INT;
    min_idx : INT;
    temp : INT;
    n : INT := 100;
    seq_local : ARRAY[1..100] OF INT;
    sort_successful : BOOL;
END_VAR

IF exe THEN
    // Initialize outputs
    error := FALSE;
    status := 16#0000;
    sort_successful := TRUE;

    // Copy input array to local working array
    FOR i := 1 TO n DO
        seq_local[i] := seq[i];
    END_FOR;

    // Selection sort algorithm
    FOR i := 1 TO n-1 DO
        min_idx := i;
        FOR j := i+1 TO n DO
            IF seq_local[j] < seq_local[min_idx] THEN
                min_idx := j;
            END_IF;
        END_FOR;

        // Swap elements if needed
        IF min_idx <> i THEN
            temp := seq_local[i];
            seq_local[i] := seq_local[min_idx];
            seq_local[min_idx] := temp;
        END_IF;
    END_FOR;

    // Copy sorted array back to output
    FOR i := 1 TO n DO
        seq[i] := seq_local[i];
    END_FOR;

    // Verify sorting was successful
    FOR i := 1 TO n-1 DO
        IF seq[i] > seq[i+1] THEN
            sort_successful := FALSE;
            EXIT;
        END_IF;
    END_FOR;

    // Set error status if verification failed
    IF NOT sort_successful THEN
        error := TRUE;
        status := 16#8A01;
    END_IF;
END_IF;

END_FUNCTION_BLOCK

(* ---- hf_6.st ---- *)
FUNCTION_BLOCK RandomNumberGenerator
VAR_INPUT
    minValue : DINT;
    maxValue : DINT;
    randomSeed_in : DINT;
END_VAR

VAR_OUTPUT
    error : BOOL;
    status : WORD;
    randomNumber : DINT;
END_VAR

VAR
    internalSeed : DINT;
END_VAR

// Initialize internal seed with provided seed
internalSeed := randomSeed_in;

// Ensure seed is positive
IF internalSeed < 0 THEN
    internalSeed := -internalSeed;
END_IF;

// Handle zero seed case
IF internalSeed = 0 THEN
    internalSeed := 1;
END_IF;

// Check for invalid range
IF minValue > maxValue THEN
    error := TRUE;
    status := 16#8200;
    randomNumber := 0;
ELSE
    // Generate random number using modulo arithmetic
    internalSeed := (internalSeed * 1103515245 + 12345) MOD 2147483647;
    randomNumber := minValue + (internalSeed MOD (maxValue - minValue + 1));

    error := FALSE;
    status := 16#0000;
END_IF;
END_FUNCTION_BLOCK

(* ---- hf_7.st ---- *)
FUNCTION_BLOCK AnalogBatchConverter
VAR_INPUT
    count : INT;
    analogValues : ARRAY[1..10] OF REAL;
END_VAR
VAR_OUTPUT
    channel_enable : ARRAY[1..10] OF BOOL;
    channel_hiLIM : ARRAY[1..10] OF REAL;
    channel_loLIM : ARRAY[1..10] OF REAL;
    channel_bipolar : ARRAY[1..10] OF BOOL;
    channel_measuringMode : ARRAY[1..10] OF INT;
    channel_retVal : ARRAY[1..10] OF WORD;
    channel_outputValue : ARRAY[1..10] OF REAL;
END_VAR
VAR
    idx : INT;
    actualCount : INT;
    rawVal : REAL;
    normalized : REAL;
    rangeSpan : REAL;
END_VAR

// Validate and limit the count parameter
actualCount := count;
IF actualCount < 1 THEN
    actualCount := 0;
ELSIF actualCount > 10 THEN
    actualCount := 10;
END_IF;

// Process each channel
FOR idx := 1 TO 10 DO
    // Initialize outputs for current channel
    channel_outputValue[idx] := 0.0;
    channel_retVal[idx] := 16#0000;

    // Only process if within active count range and enabled
    IF (idx <= actualCount) AND channel_enable[idx] THEN

        // Error Check 1: Validate measurement mode
        IF (channel_measuringMode[idx] < 0) OR (channel_measuringMode[idx] > 2) THEN
            channel_retVal[idx] := 16#8001;
            CONTINUE;
        END_IF;

        // Process based on measurement mode
        CASE channel_measuringMode[idx] OF
            0: // Non-temperature measurement
                // Error Check 2: Validate scaling limits
                IF channel_hiLIM[idx] <= channel_loLIM[idx] THEN
                    channel_retVal[idx] := 16#8002;
                    CONTINUE;
                END_IF;

                // Get raw value
                rawVal := analogValues[idx];

                // Calculate normalized value based on bipolar setting
                IF channel_bipolar[idx] THEN
                    // Bipolar: Map from -27648.0 to 27648.0
                    normalized := (rawVal + 27648.0) / 55296.0;
                ELSE
                    // Unipolar: Map from 0.0 to 27648.0
                    normalized := rawVal / 27648.0;
                END_IF;

                // Apply scaling to output range
                rangeSpan := channel_hiLIM[idx] - channel_loLIM[idx];
                channel_outputValue[idx] := channel_loLIM[idx] + (normalized * rangeSpan);

            1: // Standard temperature measurement (1/10 scaling)
                channel_outputValue[idx] := analogValues[idx] * 0.1;

            2: // Climatic temperature measurement (1/100 scaling)
                channel_outputValue[idx] := analogValues[idx] * 0.01;

        END_CASE;
    END_IF;
END_FOR;
END_FUNCTION_BLOCK

(* ---- hf_8.st ---- *)
FUNCTION_BLOCK FB_HexDigitAnalyzer
VAR_INPUT
    InputNumber: INT;
END_VAR

VAR_OUTPUT
    Thousands: INT;
    Hundreds: INT;
    Tens: INT;
    Ones: INT;
    MinDigit: INT;
    error: BOOL;
    status: WORD;
END_VAR

VAR
    tempMinValue: INT;
    tempDigit: INT;
END_VAR

METHOD FindMin: INT
VAR_INPUT
    a: INT;
    b: INT;
END_VAR
    IF a < b THEN
        FindMin := a;
    ELSE
        FindMin := b;
    END_IF;
END_METHOD

// Main execution
IF (InputNumber < 0) OR (InputNumber > 9999) THEN
    // Error condition
    error := TRUE;
    status := 16#8001;
    Thousands := 0;
    Hundreds := 0;
    Tens := 0;
    Ones := 0;
    MinDigit := 0;
ELSE
    // Valid input - process normally
    error := FALSE;
    status := 16#0000;

    // Digit separation
    Thousands := InputNumber / 1000;
    Hundreds := (InputNumber MOD 1000) / 100;
    Tens := (InputNumber MOD 100) / 10;
    Ones := InputNumber MOD 10;

    // Minimum non-zero digit detection
    tempMinValue := 32767; // Maximum INT value

    // Check thousands digit
    IF Thousands > 0 THEN
        tempMinValue := FindMin(tempMinValue, Thousands);
    END_IF;

    // Check hundreds digit
    IF Hundreds > 0 THEN
        tempMinValue := FindMin(tempMinValue, Hundreds);
    END_IF;

    // Check tens digit
    IF Tens > 0 THEN
        tempMinValue := FindMin(tempMinValue, Tens);
    END_IF;

    // Check ones digit
    IF Ones > 0 THEN
        tempMinValue := FindMin(tempMinValue, Ones);
    END_IF;

    // Set MinDigit result
    IF tempMinValue = 32767 THEN
        // All digits were zero
        MinDigit := 0;
    ELSE
        MinDigit := tempMinValue;
    END_IF;
END_IF;
END_FUNCTION_BLOCK

(* ---- hf_9.st ---- *)
FUNCTION_BLOCK ShellSortFB
VAR_INPUT
    sortDirection : BOOL; (* FALSE = Ascending, TRUE = Descending *)
    arr : ARRAY[1..1000] OF DINT;
END_VAR
VAR_OUTPUT
    error : BOOL;
    status : WORD;
    sorted_arr : ARRAY[1..1000] OF DINT;
END_VAR
VAR
    i : DINT;
    j : DINT;
    gap : DINT;
    temp : DINT;
    N : DINT := 1000;
    ascending : BOOL;
END_VAR

(* Step 1: Copy input array to output array *)
sorted_arr := arr;

(* Step 2: Initialize error outputs *)
error := FALSE;
status := 16#0000;

(* Step 3: Array size validation *)
IF N <= 1 THEN
    error := TRUE;
    status := 16#8200;
    RETURN;
END_IF;

IF N > 1000 THEN
    error := TRUE;
    status := 16#8201;
    RETURN;
END_IF;

(* Step 4: Determine sorting direction *)
ascending := NOT sortDirection; (* TRUE for ascending, FALSE for descending *)

(* Step 5: Shell Sort Algorithm *)
gap := N / 2;

WHILE gap > 0 DO
    i := gap + 1;

    WHILE i <= N DO
        temp := sorted_arr[i];
        j := i;

        WHILE (j > gap) AND (
            (ascending AND (sorted_arr[j - gap] > temp)) OR
            (NOT ascending AND (sorted_arr[j - gap] < temp))
        ) DO
            sorted_arr[j] := sorted_arr[j - gap];
            j := j - gap;
        END_WHILE;

        sorted_arr[j] := temp;
        i := i + 1;
    END_WHILE;

    gap := gap / 2;
END_WHILE;

(* Step 6: Final status setting (already set to success at initialization) *)
END_FUNCTION_BLOCK

(* ---- med_22.st ---- *)
FUNCTION_BLOCK CottonCandyMachine
VAR_INPUT
    SugarLevel : REAL; (* Input for sugar level *)
    SpinningSpeed : INT; (* Input for spinning speed *)
END_VAR
VAR_OUTPUT
    SugarFeeder : BOOL; (* Output to control sugar feeding *)
    MotorSpeed : INT; (* Output to control spinning motor speed *)
END_VAR

// Main logic
IF SugarLevel < 10.0 THEN
    SugarFeeder := TRUE;
ELSE
    SugarFeeder := FALSE;
END_IF;

IF SpinningSpeed > 0 THEN
    MotorSpeed := SpinningSpeed;
ELSE
    MotorSpeed := 0;
END_IF;

END_FUNCTION_BLOCK

(* ---- med_23.st ---- *)
FUNCTION_BLOCK SmartIrrigationSystem
VAR_INPUT
    SoilMoistureSensor1 : REAL;
    SoilMoistureSensor2 : REAL;
    WeatherForecast : INT; (* 0: Sunny, 1: Rainy, 2: Cloudy *)
END_VAR

VAR_OUTPUT
    WaterPump : BOOL;
END_VAR

VAR
    SoilMoistureThreshold : REAL := 30.0;
END_VAR

(* Main irrigation logic *)
IF WeatherForecast = 1 THEN
    (* Priority: Deactivate pump immediately if rain is forecast *)
    WaterPump := FALSE;
ELSIF WeatherForecast = 0 THEN
    (* Sunny weather: Activate pump if at least one sensor is below threshold *)
    IF (SoilMoistureSensor1 < SoilMoistureThreshold) OR (SoilMoistureSensor2 < SoilMoistureThreshold) THEN
        WaterPump := TRUE;
    ELSE
        WaterPump := FALSE;
    END_IF;
ELSE
    (* Cloudy or other weather conditions: Keep pump off *)
    WaterPump := FALSE;
END_IF;

END_FUNCTION_BLOCK

(* ---- med_24.st ---- *)
FUNCTION_BLOCK AutomaticDoorControl
VAR_INPUT
    ProximitySensor : BOOL;
    ElapsedTime : DINT; (* Time since door was last opened in milliseconds *)
END_VAR

VAR_OUTPUT
    DoorOpen : BOOL;
END_VAR

VAR
    DoorOpenDuration : DINT := 5000; (* 5 seconds in milliseconds *)
    eState : (eDoorClosed, eDoorOpening, eDoorOpen, eDoorClosing) := eDoorClosed;
    rTrigSensor : R_TRIG;
    fTrigSensor : F_TRIG;
    tDoorTimer : TON;
    bTimerStarted : BOOL := FALSE;
    bProxPrev : BOOL := FALSE;
END_VAR

(* Detect rising and falling edges of proximity sensor *)
rTrigSensor(CLK := ProximitySensor);
fTrigSensor(CLK := ProximitySensor);

CASE eState OF
    eDoorClosed:
        DoorOpen := FALSE;
        bTimerStarted := FALSE;
        tDoorTimer(IN := FALSE);

        (* Open door when proximity sensor detects object *)
        IF rTrigSensor.Q THEN
            eState := eDoorOpening;
        END_IF;

    eDoorOpening:
        DoorOpen := TRUE;
        (* Start timer for door open duration *)
        tDoorTimer(IN := TRUE, PT := DINT_TO_TIME(DoorOpenDuration));
        bTimerStarted := TRUE;
        eState := eDoorOpen;

    eDoorOpen:
        DoorOpen := TRUE;

        (* Keep timer running while door is open *)
        IF bTimerStarted THEN
            tDoorTimer(IN := TRUE);
        END_IF;

        (* Close door if proximity sensor becomes inactive OR timer expires *)
        IF fTrigSensor.Q OR tDoorTimer.Q THEN
            eState := eDoorClosing;
            tDoorTimer(IN := FALSE);
            bTimerStarted := FALSE;
        END_IF;

    eDoorClosing:
        DoorOpen := FALSE;
        tDoorTimer(IN := FALSE);
        bTimerStarted := FALSE;

        (* Wait for elapsed time before allowing next open cycle *)
        (* This prevents rapid open/close cycles *)
        IF ElapsedTime >= 1000 THEN (* 1 second cooldown *)
            eState := eDoorClosed;
        END_IF;
END_CASE;

(* Store previous proximity sensor state for edge detection *)
bProxPrev := ProximitySensor;
END_FUNCTION_BLOCK

(* ---- med_25.st ---- *)
FUNCTION_BLOCK WastewaterControl
VAR_INPUT
    InFlow : REAL;
    OutFlow : REAL;
    pH : REAL;
    TankLvl : REAL;
END_VAR

VAR_OUTPUT
    Pump1 : BOOL;
    Pump2 : BOOL;
    Valve1 : BOOL;
    Valve2 : BOOL;
END_VAR

VAR
    LowInFlow : REAL := 100.0;
    HighOutFlow : REAL := 90.0;
    DesiredPH : REAL := 7.0;
    HighTankLvl : REAL := 80.0;
END_VAR

// Control logic implementation
Pump1 := (InFlow < LowInFlow);
Pump2 := (OutFlow > HighOutFlow);
Valve1 := (pH < DesiredPH);
Valve2 := (TankLvl > HighTankLvl);

END_FUNCTION_BLOCK

(* ---- med_26.st ---- *)
FUNCTION_BLOCK BookSorting
VAR_INPUT
    RFID1 : BOOL;
    RFID2 : BOOL;
    RFID3 : BOOL;
END_VAR

VAR_OUTPUT
    Motor : BOOL;
    Bin1 : BOOL;
    Bin2 : BOOL;
    Bin3 : BOOL;
END_VAR

// Implementation
Motor := RFID1 OR RFID2 OR RFID3;

IF RFID1 THEN
    Bin1 := TRUE;
    Bin2 := FALSE;
    Bin3 := FALSE;
ELSIF RFID2 THEN
    Bin1 := FALSE;
    Bin2 := TRUE;
    Bin3 := FALSE;
ELSIF RFID3 THEN
    Bin1 := FALSE;
    Bin2 := FALSE;
    Bin3 := TRUE;
ELSE
    Bin1 := FALSE;
    Bin2 := FALSE;
    Bin3 := FALSE;
END_IF;

END_FUNCTION_BLOCK

(* ---- med_27.st ---- *)
FUNCTION_BLOCK FlowerArrangingMachine
VAR_INPUT
    FlowerTypeSensor : INT; (* Input for detecting flower type *)
    FlowerColorSensor : INT; (* Input for detecting flower color *)
END_VAR
VAR_OUTPUT
    ArrangingMechanism : INT; (* Output for controlling arranging mechanism *)
    ConveyorBelt : BOOL; (* Output for controlling conveyor belt *)
END_VAR

(* Main control logic *)
IF (FlowerTypeSensor = 1) AND (FlowerColorSensor = 1) THEN
    ArrangingMechanism := 1;
ELSIF (FlowerTypeSensor = 1) AND (FlowerColorSensor = 2) THEN
    ArrangingMechanism := 2;
ELSIF (FlowerTypeSensor = 2) AND (FlowerColorSensor = 1) THEN
    ArrangingMechanism := 3;
ELSIF (FlowerTypeSensor = 2) AND (FlowerColorSensor = 2) THEN
    ArrangingMechanism := 4;
ELSE
    ArrangingMechanism := 0;
END_IF;

(* Conveyor belt control based on arranging mechanism *)
ConveyorBelt := (ArrangingMechanism <> 0);

END_FUNCTION_BLOCK

(* ---- med_28.st ---- *)
FUNCTION_BLOCK HomeBrewingSystem
VAR_INPUT
    TemperatureSensor : REAL; (* Input for temperature measurement *)
    WaterFlowSensor : REAL; (* Input for water flow measurement *)
    BrewingStartTime : TIME; (* Input for brewing start time *)
    BrewingDuration : TIME; (* Input for brewing duration *)
END_VAR
VAR_OUTPUT
    HeatingElement : BOOL; (* Output for heating element *)
    AgitationMotor : BOOL; (* Output for agitation motor *)
    HopsDispenser : BOOL; (* Output for hops dispenser *)
    FermentationTank : BOOL; (* Output for fermentation tank *)
END_VAR
VAR
    CurrentTime : TIME;
    ElapsedBrewingTime : TIME;
    TemperatureSetpoint : REAL := 65.0;
    FlowThreshold : REAL := 0.5;
    HopsDispenseTime : TIME := T#5h;
    FermentationStartTime : TIME := T#48h;
END_VAR

    (* Calculate current time and elapsed brewing time *)
    CurrentTime := TIME();
    ElapsedBrewingTime := CurrentTime - BrewingStartTime;

    (* Control Heating Element based on temperature *)
    IF TemperatureSensor < TemperatureSetpoint THEN
        HeatingElement := TRUE;
    ELSE
        HeatingElement := FALSE;
    END_IF;

    (* Control Agitation Motor based on water flow *)
    IF WaterFlowSensor > FlowThreshold THEN
        AgitationMotor := TRUE;
    ELSE
        AgitationMotor := FALSE;
    END_IF;

    (* Control Hops Dispenser after 5 hours of brewing *)
    IF ElapsedBrewingTime >= HopsDispenseTime THEN
        HopsDispenser := TRUE;
    ELSE
        HopsDispenser := FALSE;
    END_IF;

    (* Control Fermentation Tank after 48 hours of brewing *)
    IF ElapsedBrewingTime >= FermentationStartTime THEN
        FermentationTank := TRUE;
    ELSE
        FermentationTank := FALSE;
    END_IF;

END_FUNCTION_BLOCK

(* ---- med_29.st ---- *)
FUNCTION_BLOCK DocumentFilingSystem
VAR_INPUT
    DocumentInlet : BOOL; (* Input to detect the arrival of a document *)
    CategorySelector : INT; (* Input to select the document category *)
END_VAR
VAR_OUTPUT
    ConveyorMotor : BOOL; (* Output to control the conveyor motor *)
    StorageBin1 : BOOL; (* Output to activate storage bin 1 *)
    StorageBin2 : BOOL; (* Output to activate storage bin 2 *)
    StorageBin3 : BOOL; (* Output to activate storage bin 3 *)
    StorageBin4 : BOOL; (* Output to activate storage bin 4 *)
END_VAR
VAR
    ValidCategory : BOOL; (* Internal flag for valid category range *)
END_VAR

(* Check if category selector is within valid range (1-4) *)
ValidCategory := (CategorySelector >= 1) AND (CategorySelector <= 4);

(* Main control logic *)
IF DocumentInlet AND ValidCategory THEN
    (* Activate conveyor motor when document is present and category is valid *)
    ConveyorMotor := TRUE;

    (* Activate only the selected storage bin based on category *)
    CASE CategorySelector OF
        1:
            StorageBin1 := TRUE;
            StorageBin2 := FALSE;
            StorageBin3 := FALSE;
            StorageBin4 := FALSE;
        2:
            StorageBin1 := FALSE;
            StorageBin2 := TRUE;
            StorageBin3 := FALSE;
            StorageBin4 := FALSE;
        3:
            StorageBin1 := FALSE;
            StorageBin2 := FALSE;
            StorageBin3 := TRUE;
            StorageBin4 := FALSE;
        4:
            StorageBin1 := FALSE;
            StorageBin2 := FALSE;
            StorageBin3 := FALSE;
            StorageBin4 := TRUE;
        ELSE
            (* This should never happen since ValidCategory is checked, but included for safety *)
            StorageBin1 := FALSE;
            StorageBin2 := FALSE;
            StorageBin3 := FALSE;
            StorageBin4 := FALSE;
    END_CASE;
ELSE
    (* Deactivate all outputs when no document or invalid category *)
    ConveyorMotor := FALSE;
    StorageBin1 := FALSE;
    StorageBin2 := FALSE;
    StorageBin3 := FALSE;
    StorageBin4 := FALSE;
END_IF;

END_FUNCTION_BLOCK

(* ---- med_30.st ---- *)
FUNCTION_BLOCK MuseumClimateControl
VAR_INPUT
    HumiditySensor : REAL;
    TemperatureSensor : REAL;
    LightSensor : BOOL;
END_VAR

VAR_OUTPUT
    HVACSystem : BOOL;
    Humidifier : BOOL;
    Dehumidifier : BOOL;
    LightControl : BOOL;
END_VAR

VAR
    TargetHumidity : REAL := 50.0;
    TargetTemperature : REAL := 20.0;
    LightThreshold : BOOL := TRUE;
END_VAR

// Humidity control logic
Humidifier := FALSE;
Dehumidifier := FALSE;

IF HumiditySensor < TargetHumidity THEN
    Humidifier := TRUE;
ELSIF HumiditySensor > TargetHumidity THEN
    Dehumidifier := TRUE;
END_IF;

// Temperature control logic
IF TemperatureSensor <> TargetTemperature THEN
    HVACSystem := TRUE;
ELSE
    HVACSystem := FALSE;
END_IF;

// Lighting control logic
IF LightSensor AND LightThreshold THEN
    LightControl := FALSE;  // Turn off lights when bright
ELSE
    LightControl := TRUE;   // Turn on lights otherwise
END_IF;

END_FUNCTION_BLOCK

(* ---- med_31.st ---- *)
FUNCTION_BLOCK ChargingStationControl
VAR_INPUT
    EVConnected : BOOL;
    EVVoltage : REAL;
    EVCurrent : REAL;
    EVStateOfCharge : REAL;
    ChargingTimer : TIME;
END_VAR

VAR_OUTPUT
    EVCharging : BOOL;
END_VAR

VAR
    VoltageOK : BOOL;
    CurrentOK : BOOL;
    SOCNotFull : BOOL;
    TimerOK : BOOL;
END_VAR

(* Evaluate individual conditions *)
VoltageOK := EVVoltage > 350.0;
CurrentOK := EVCurrent <= 32.0;
SOCNotFull := EVStateOfCharge < 100.0;
TimerOK := ChargingTimer <= T#2h;

(* Control charging output based on all conditions *)
IF EVConnected AND VoltageOK AND CurrentOK AND SOCNotFull AND TimerOK THEN
    EVCharging := TRUE;
ELSE
    EVCharging := FALSE;
END_IF

END_FUNCTION_BLOCK

(* ---- med_32.st ---- *)
FUNCTION_BLOCK GreenhouseWateringSystem
VAR_INPUT
    SoilMoistureSensor : REAL;   (* Input for soil moisture level (0-100%) *)
END_VAR

VAR_OUTPUT
    SprinklersOn : BOOL := FALSE; (* Output for controlling sprinklers - on/off *)
END_VAR

VAR
    ResponseDelay : TIME := T#5s;  (* Response delay for the system *)
    TransitionTimer : TON;         (* Timer for managing state transitions *)
    EnableDelay : BOOL := FALSE;   (* Flag to enable delay timing *)
    LastMoistureReading : REAL := 100.0; (* Initialize to ensure sprinklers start off *)
END_VAR

(* Main control logic *)
TransitionTimer(IN:=EnableDelay, PT:=ResponseDelay);

(* Store current moisture reading for next cycle *)
LastMoistureReading := SoilMoistureSensor;

(* Control logic with response delay consideration *)
IF NOT TransitionTimer.Q THEN
    (* Timer is running - wait for delay before changing state *)
    IF TransitionTimer.IN THEN
        (* Continue timing, no state change yet *)
        SprinklersOn := SprinklersOn; (* Maintain current state *)
    ELSE
        (* No transition pending - evaluate conditions *)
        IF (NOT SprinklersOn) AND (SoilMoistureSensor < 30.0) THEN
            (* Condition met to turn sprinklers ON - start delay timer *)
            EnableDelay := TRUE;
        ELSIF SprinklersOn AND (SoilMoistureSensor > 70.0) THEN
            (* Condition met to turn sprinklers OFF - start delay timer *)
            EnableDelay := TRUE;
        ELSE
            (* No transition needed - ensure timer is not running *)
            EnableDelay := FALSE;
            TransitionTimer(IN:=FALSE); (* Reset timer *)
        END_IF;
    END_IF;
ELSE
    (* Timer has completed - execute state transition *)
    EnableDelay := FALSE; (* Reset enable flag *)
    TransitionTimer(IN:=FALSE); (* Reset timer *)

    (* Determine which transition to execute based on last evaluation *)
    IF (NOT SprinklersOn) AND (LastMoistureReading < 30.0) THEN
        SprinklersOn := TRUE;
    ELSIF SprinklersOn AND (LastMoistureReading > 70.0) THEN
        SprinklersOn := FALSE;
    END_IF;
END_IF;
END_FUNCTION_BLOCK

(* ---- med_33.st ---- *)
FUNCTION_BLOCK RoboticArmColorSorting
VAR_INPUT
    ColorSensorRed : BOOL;   (* Input: Red color sensor *)
    ColorSensorGreen : BOOL;  (* Input: Green color sensor *)
    ColorSensorBlue : BOOL;   (* Input: Blue color sensor *)
END_VAR

VAR_OUTPUT
    RoboticArmMove : BOOL := FALSE;     (* Output: Control for robotic arm movement *)
    BinRed : BOOL := FALSE;           (* Output: Activate red bin *)
    BinGreen : BOOL := FALSE;         (* Output: Activate green bin *)
    BinBlue : BOOL := FALSE;          (* Output: Activate blue bin *)
END_VAR

(* Main logic *)
RoboticArmMove := ColorSensorRed OR ColorSensorGreen OR ColorSensorBlue;

(* Exclusive bin activation with priority: Red > Green > Blue *)
BinRed := ColorSensorRed;
BinGreen := ColorSensorGreen AND NOT ColorSensorRed;
BinBlue := ColorSensorBlue AND NOT ColorSensorRed AND NOT ColorSensorGreen;

END_FUNCTION_BLOCK

(* ---- med_34.st ---- *)
FUNCTION_BLOCK CoffeeMachineControl
VAR_INPUT
    StartButton : BOOL;
    ElapsedTime : DINT; (* Time elapsed since the start of the current process, in milliseconds *)
END_VAR

VAR_OUTPUT
    WaterHeating : BOOL;
    GrinderRunning : BOOL;
    Brewing : BOOL;
    WaterHeated : BOOL;
    GrinderFinished : BOOL;
    CoffeeReady : BOOL;
END_VAR

VAR
    WaterHeatingDuration : DINT := 30000; (* 30 seconds in milliseconds *)
    GrinderDuration : DINT := 15000; (* 15 seconds in milliseconds *)
    BrewingDuration : DINT := 60000; (* 60 seconds in milliseconds *)
    CurrentState : INT := 0;
    ProcessStartTime : DINT := 0;
END_VAR

(* Reset all outputs when start button is not pressed *)
IF NOT StartButton THEN
    CurrentState := 0;
    ProcessStartTime := 0;
    WaterHeating := FALSE;
    GrinderRunning := FALSE;
    Brewing := FALSE;
    WaterHeated := FALSE;
    GrinderFinished := FALSE;
    CoffeeReady := FALSE;
ELSE
    CASE CurrentState OF
        0: (* Idle - waiting for start *)
            WaterHeating := FALSE;
            GrinderRunning := FALSE;
            Brewing := FALSE;
            WaterHeated := FALSE;
            GrinderFinished := FALSE;
            CoffeeReady := FALSE;

            IF StartButton THEN
                WaterHeating := TRUE;
                ProcessStartTime := ElapsedTime;
                CurrentState := 1;
            END_IF;

        1: (* Water Heating *)
            WaterHeating := TRUE;
            GrinderRunning := FALSE;
            Brewing := FALSE;

            IF (ElapsedTime - ProcessStartTime) >= WaterHeatingDuration THEN
                WaterHeating := FALSE;
                WaterHeated := TRUE;
                ProcessStartTime := ElapsedTime;
                CurrentState := 2;
            END_IF;

        2: (* Grinder Running *)
            WaterHeating := FALSE;
            GrinderRunning := TRUE;
            Brewing := FALSE;

            IF (ElapsedTime - ProcessStartTime) >= GrinderDuration THEN
                GrinderRunning := FALSE;
                GrinderFinished := TRUE;
                ProcessStartTime := ElapsedTime;
                CurrentState := 3;
            END_IF;

        3: (* Brewing *)
            WaterHeating := FALSE;
            GrinderRunning := FALSE;
            Brewing := TRUE;

            IF (ElapsedTime - ProcessStartTime) >= BrewingDuration THEN
                Brewing := FALSE;
                CoffeeReady := TRUE;
                CurrentState := 4;
            END_IF;

        4: (* Process Complete *)
            WaterHeating := FALSE;
            GrinderRunning := FALSE;
            Brewing := FALSE;
            (* Keep status indicators active until reset *)

        ELSE
            CurrentState := 0;
    END_CASE;
END_IF;

END_FUNCTION_BLOCK

(* ---- med_35.st ---- *)
FUNCTION_BLOCK FB_SimpleCalculation
VAR_INPUT
    INPUT_VAR1 : INT := 2;
    VAR2 : INT := 0;
END_VAR
VAR_OUTPUT
    OUTPUT_VAR1 : INT;
    OUTPUT_VAR2 : INT;
END_VAR
VAR
    i : INT;
    tempVar1 : INT;
    tempVar2 : INT;
END_VAR

// First calculation: Multiply INPUT_VAR1 by 2 for 5 iterations
tempVar1 := INPUT_VAR1;
FOR i := 1 TO 5 DO
    tempVar1 := tempVar1 * 2;
END_FOR;
OUTPUT_VAR1 := tempVar1;

// Second calculation: Increment VAR2 by 1 for 5 iterations
tempVar2 := VAR2;
FOR i := 1 TO 5 DO
    tempVar2 := tempVar2 + 1;
END_FOR;
OUTPUT_VAR2 := tempVar2;

END_FUNCTION_BLOCK

(* ---- med_36.st ---- *)
FUNCTION_BLOCK FB_ExpandedPoint
    VAR_INPUT
        INPUT_VAR2 : INT;
        INPUT_VAR1_X : INT;
        INPUT_VAR1_Y : INT;
        INPUT_VAR3_X : INT := 1;
        INPUT_VAR3_Y : INT := 2;
    END_VAR

    VAR_OUTPUT
        OUTPUT_VAR2 : INT;
        OUTPUT_VAR1_X : INT;
        OUTPUT_VAR1_Y : INT;
        OUTPUT_VAR3_X : INT;
        OUTPUT_VAR3_Y : INT;
    END_VAR

    // Main execution logic
    OUTPUT_VAR2 := INPUT_VAR2;
    OUTPUT_VAR1_X := 1;
    OUTPUT_VAR1_Y := 2;
    OUTPUT_VAR3_X := 100;
    OUTPUT_VAR3_Y := -7000;
END_FUNCTION_BLOCK

(* ---- med_37.st ---- *)
FUNCTION_BLOCK FB_RealValueAdjuster
VAR_INPUT
    x_in : REAL;
END_VAR
VAR_OUTPUT
    x_out : REAL;
END_VAR
VAR
    x_temp : REAL;
    int_val : INT;
END_VAR

// Initialize with input value
x_temp := x_in;

// First condition: if input is exactly 0.0, add 1.0
IF x_in = 0.0 THEN
    x_temp := x_temp + 1.0;
END_IF;

// Second condition: if input is not 0.0, also add 1.0
IF x_in <> 0.0 THEN
    x_temp := x_temp + 1.0;
END_IF;

// Third condition: convert to integer and check
int_val := REAL_TO_INT(x_in);
IF int_val <> 0 THEN
    x_temp := x_temp + 1.0;
END_IF;

// Assign final result to output
x_out := x_temp;

END_FUNCTION_BLOCK

(* ---- med_38.st ---- *)
FUNCTION_BLOCK SolarPanelTracking
VAR_INPUT
    SolarIntensity : REAL;      (* Input: Solar intensity in percentage *)
    CurrentTime : TIME;         (* Input: Current time of day *)
END_VAR

VAR_OUTPUT
    PanelAngle : REAL := 0.0;   (* Output: Panel angle in degrees *)
END_VAR

VAR
    SunriseTime : TIME := T#6H;    (* Sunrise time set to 6 AM *)
    SunsetTime : TIME := T#18H;    (* Sunset time set to 6 PM *)
    NoonTime : TIME := T#12H;      (* Noon time set to 12 PM *)
    MorningAngle : REAL := 30.0;   (* Angle during morning *)
    NoonAngle : REAL := 60.0;      (* Angle during noon *)
    EveningAngle : REAL := 30.0;   (* Angle during evening *)

    eState : (STATE_NIGHT, STATE_MORNING, STATE_NOON, STATE_EVENING);
END_VAR

(* Determine state based on time and solar intensity *)
IF (CurrentTime < SunriseTime) OR (CurrentTime >= SunsetTime) THEN
    eState := STATE_NIGHT;
ELSIF SolarIntensity >= 90.0 THEN
    eState := STATE_NOON;
ELSIF CurrentTime < NoonTime THEN
    eState := STATE_MORNING;
ELSE
    eState := STATE_EVENING;
END_IF;

(* Set panel angle based on state *)
CASE eState OF
    STATE_NIGHT:
        PanelAngle := 0.0;
    STATE_MORNING:
        PanelAngle := MorningAngle;
    STATE_NOON:
        PanelAngle := NoonAngle;
    STATE_EVENING:
        PanelAngle := EveningAngle;
END_CASE;

(* Ensure panel angle is within 0 to 90 degrees *)
IF PanelAngle < 0.0 THEN
    PanelAngle := 0.0;
ELSIF PanelAngle > 90.0 THEN
    PanelAngle := 90.0;
END_IF;

END_FUNCTION_BLOCK

(* ---- med_39.st ---- *)
FUNCTION_BLOCK WindTurbineControl
VAR_INPUT
    WindSpeedSensor : REAL; (* Input for measuring wind speed *)
    GeneratorSpeedSensor : REAL; (* Input for measuring generator speed *)
END_VAR

VAR_OUTPUT
    BladePitch : INT; (* Output for blade pitch control (degrees) *)
    GeneratorSpeed : REAL; (* Output for generator speed control (RPM) *)
END_VAR

(* Main control logic *)
IF WindSpeedSensor <= 3.0 THEN
    (* Low wind speed condition *)
    BladePitch := -5;
    GeneratorSpeed := 500.0;
ELSIF (WindSpeedSensor > 3.0) AND (WindSpeedSensor <= 5.0) THEN
    (* Moderate wind speed condition *)
    BladePitch := 0;
    GeneratorSpeed := 800.0;
ELSIF WindSpeedSensor > 5.0 THEN
    (* High wind speed condition *)
    BladePitch := 5;
    GeneratorSpeed := 1000.0;
ELSE
    (* Fallback condition for invalid inputs *)
    BladePitch := 0;
    GeneratorSpeed := 0.0;
END_IF;

END_FUNCTION_BLOCK

(* ---- med_40.st ---- *)
FUNCTION_BLOCK RockClimbingWallControl
VAR_INPUT
    UserWeightSensor : REAL; (* Input for measuring the user's weight *)
    WallDifficultyLevel : INT; (* Input for setting the wall's initial difficulty level *)
    WallHeight : REAL; (* Input for setting the wall's height *)
    RouteSelector : INT; (* Input for selecting a climbing route *)
END_VAR
VAR_OUTPUT
    ClimbingMotorSpeed : REAL; (* Output for controlling the climbing wall motor speed *)
    WallLights : BOOL; (* Output for controlling wall lighting *)
END_VAR

VAR
    internalDifficultyLevel : INT; (* Internal variable for calculated difficulty level *)
END_VAR

(* Main execution logic *)

(* Set difficulty level based on route selector *)
CASE RouteSelector OF
    1: internalDifficultyLevel := 1;
    2: internalDifficultyLevel := 2;
    3: internalDifficultyLevel := 3;
    ELSE
        (* Fallback to input difficulty level if route selector is invalid *)
        internalDifficultyLevel := WallDifficultyLevel;
END_CASE;

(* Adjust climbing motor speed based on user weight *)
IF UserWeightSensor > 60.0 THEN
    ClimbingMotorSpeed := 1.0;
ELSE
    ClimbingMotorSpeed := 0.8;
END_IF;

(* Control wall lights based on wall height *)
IF WallHeight > 5.0 THEN
    WallLights := TRUE;
ELSE
    WallLights := FALSE;
END_IF;

END_FUNCTION_BLOCK

(* ---- med_41.st ---- *)
FUNCTION_BLOCK FishTankControl
VAR_INPUT
    OxygenLevel : REAL; (* Input for oxygen level in the tank *)
    WaterTemperature : REAL; (* Input for water temperature *)
    FeedingTime : TIME; (* Time for scheduled feeding *)
    CurrentTime : TIME; (* Current system time *)
END_VAR
VAR_OUTPUT
    OxygenValve : BOOL; (* Output to control oxygen supply *)
    Heater : BOOL; (* Output to control the heater *)
    Feeder : BOOL; (* Output to control the fish feeder *)
END_VAR

// Main logic implementation
IF OxygenLevel < 5.0 THEN
    OxygenValve := TRUE;
ELSE
    OxygenValve := FALSE;
END_IF;

IF WaterTemperature < 25.0 THEN
    Heater := TRUE;
ELSE
    Heater := FALSE;
END_IF;

IF CurrentTime >= FeedingTime THEN
    Feeder := TRUE;
ELSE
    Feeder := FALSE;
END_IF;

END_FUNCTION_BLOCK

(* ---- med_42.st ---- *)
FUNCTION_BLOCK RetractableRoofControl
VAR_INPUT
    RainSensor : BOOL; (* Input to detect rain *)
    WindSensor : BOOL; (* Input to detect wind *)
    TemperatureSensor : REAL; (* Input to measure temperature *)
END_VAR
VAR_OUTPUT
    RoofMotor : BOOL; (* Output to control the roof motor *)
END_VAR

// Main control logic
IF RainSensor AND WindSensor THEN
    RoofMotor := FALSE; (* Close completely *)
ELSIF RainSensor AND NOT WindSensor THEN
    RoofMotor := TRUE; (* Partially close *)
ELSIF NOT RainSensor AND TemperatureSensor < 20.0 THEN
    RoofMotor := TRUE; (* Close slightly *)
ELSIF NOT RainSensor AND TemperatureSensor >= 20.0 THEN
    RoofMotor := FALSE; (* Fully open *)
ELSE
    RoofMotor := FALSE; (* Default safe state *)
END_IF;

END_FUNCTION_BLOCK

(* ---- med_43.st ---- *)
FUNCTION_BLOCK SandwichMaker
VAR_INPUT
    BreadFeeder : BOOL; (* Input: Detects the presence of bread slices *)
    Ingredient1 : BOOL; (* Input: Detects the presence of Ingredient 1 (e.g., cheese) *)
    Ingredient2 : BOOL; (* Input: Detects the presence of Ingredient 2 (e.g., lettuce) *)
    Ingredient3 : BOOL; (* Input: Detects the presence of Ingredient 3 (e.g., tomatoes) *)
    Condiment1 : BOOL; (* Input: Detects the presence of Condiment 1 (e.g., mayo) *)
    Condiment2 : BOOL; (* Input: Detects the presence of Condiment 2 (e.g., mustard) *)
END_VAR
VAR_OUTPUT
    ConveyorMotor : BOOL; (* Output: Controls the conveyor belt motor *)
    AssembleMotor : BOOL; (* Output: Controls the sandwich assembly motor *)
END_VAR
VAR
    SliceCount : INT := 0; (* Counter for bread slices *)
    BreadFeederPrev : BOOL := FALSE; (* Previous state for edge detection *)
END_VAR

(* Conveyor motor control and slice counting *)
IF BreadFeeder THEN
    ConveyorMotor := TRUE;

    (* Count bread slices on rising edge *)
    IF NOT BreadFeederPrev THEN
        SliceCount := SliceCount + 1;
    END_IF;
ELSE
    ConveyorMotor := FALSE;
END_IF;

(* Store current BreadFeeder state for next cycle *)
BreadFeederPrev := BreadFeeder;

(* Assembly motor control *)
IF (SliceCount >= 2) AND
   Ingredient1 AND Ingredient2 AND Ingredient3 AND
   Condiment1 AND Condiment2 THEN
    AssembleMotor := TRUE;
ELSE
    AssembleMotor := FALSE;
END_IF;

END_FUNCTION_BLOCK

(* ---- med_44.st ---- *)
FUNCTION_BLOCK DroneChargingStation
VAR_INPUT
    Drone1BatteryLevel : INT := 0; (* Battery level of Drone 1 (0-100%) *)
    Drone2BatteryLevel : INT := 0; (* Battery level of Drone 2 (0-100%) *)
    Drone3BatteryLevel : INT := 0; (* Battery level of Drone 3 (0-100%) *)
    ChargingTime : TIME := T#30s; (* Charging time required for each drone *)
END_VAR
VAR_OUTPUT
    Drone1Status : BOOL := FALSE; (* Status of Drone 1 *)
    Drone2Status : BOOL := FALSE; (* Status of Drone 2 *)
    Drone3Status : BOOL := FALSE; (* Status of Drone 3 *)
    ChargingStationStatus : BOOL := FALSE; (* Charging station status *)
    DroneDeployed : BOOL := FALSE; (* Indicates if a drone is deployed *)
END_VAR
VAR
    TimeRemaining : TIME := T#0s; (* Remaining charging time for the current charging operation *)
    ChargingDrone : INT := 0; (* 0 = none, 1 = drone1, 2 = drone2, 3 = drone3 *)
    TimerActive : BOOL := FALSE; (* Timer activation flag *)
END_VAR

(* Deployment recall logic - check if any drone battery falls below 10% *)
IF DroneDeployed THEN
    IF (Drone1BatteryLevel < 10) OR (Drone2BatteryLevel < 10) OR (Drone3BatteryLevel < 10) THEN
        DroneDeployed := FALSE;
    END_IF;
END_IF;

(* Charging station management logic *)
IF NOT ChargingStationStatus THEN
    (* Station is free - check for drones needing charge *)
    Drone1Status := FALSE;
    Drone2Status := FALSE;
    Drone3Status := FALSE;
    TimerActive := FALSE;

    IF ChargingDrone = 0 THEN
        (* Select first drone with battery below 20% *)
        IF (Drone1BatteryLevel < 20) AND (Drone1BatteryLevel >= 0) THEN
            ChargingDrone := 1;
            TimeRemaining := ChargingTime;
        ELSIF (Drone2BatteryLevel < 20) AND (Drone2BatteryLevel >= 0) THEN
            ChargingDrone := 2;
            TimeRemaining := ChargingTime;
        ELSIF (Drone3BatteryLevel < 20) AND (Drone3BatteryLevel >= 0) THEN
            ChargingDrone := 3;
            TimeRemaining := ChargingTime;
        END_IF;
    END_IF;

    (* Start charging if a drone is selected *)
    IF ChargingDrone > 0 THEN
        ChargingStationStatus := TRUE;
        TimerActive := TRUE;

        CASE ChargingDrone OF
            1: Drone1Status := TRUE;
            2: Drone2Status := TRUE;
            3: Drone3Status := TRUE;
        END_CASE;
    END_IF;
ELSE
    (* Station is busy - handle charging timer *)
    IF TimerActive THEN
        IF TimeRemaining > T#0s THEN
            TimeRemaining := TimeRemaining - T#1ms; (* Decrement timer - adjust cycle time as needed *)
        ELSE
            (* Charging complete *)
            Drone1Status := FALSE;
            Drone2Status := FALSE;
            Drone3Status := FALSE;
            ChargingStationStatus := FALSE;
            ChargingDrone := 0;
            TimerActive := FALSE;
            TimeRemaining := T#0s;
        END_IF;
    END_IF;
END_IF;

END_FUNCTION_BLOCK

(* ---- med_45.st ---- *)
FUNCTION_BLOCK AutomatedSmoothieMaker
VAR_INPUT
    BananaAvailable : BOOL;
    BerryMixAvailable : BOOL;
    SpinachAvailable : BOOL;
    YogurtAvailable : BOOL;
    CustomerPreference : INT;
END_VAR

VAR_OUTPUT
    BlenderMotor : BOOL;
    Dispenser : BOOL;
END_VAR

VAR
    RecipeValid : BOOL;
    IngredientsAvailable : BOOL;
END_VAR

// Initialize outputs and internal variables
BlenderMotor := FALSE;
Dispenser := FALSE;
RecipeValid := FALSE;
IngredientsAvailable := FALSE;

// Determine recipe validity and ingredient availability based on customer preference
CASE CustomerPreference OF
    1: // Recipe 1: Banana, Berry Mix, Yogurt
        RecipeValid := TRUE;
        IngredientsAvailable := BananaAvailable AND BerryMixAvailable AND YogurtAvailable;

    2: // Recipe 2: Berry Mix, Spinach, Yogurt
        RecipeValid := TRUE;
        IngredientsAvailable := BerryMixAvailable AND SpinachAvailable AND YogurtAvailable;

    3: // Recipe 3: Banana, Spinach, Yogurt
        RecipeValid := TRUE;
        IngredientsAvailable := BananaAvailable AND SpinachAvailable AND YogurtAvailable;

    ELSE
        // Invalid preference
        RecipeValid := FALSE;
        IngredientsAvailable := FALSE;
END_CASE;

// Control blender motor and dispenser based on recipe validity and ingredient availability
IF RecipeValid AND IngredientsAvailable THEN
    Dispenser := TRUE;
    BlenderMotor := TRUE;
ELSE
    Dispenser := FALSE;
    BlenderMotor := FALSE;
END_IF;

END_FUNCTION_BLOCK

(* ---- med_46.st ---- *)
FUNCTION_BLOCK PrecisionEngravingMachine
VAR_INPUT
    DesignSelection : INT;
    EngravingDepth : REAL;
    EngravingSpeed : REAL;
END_VAR

VAR_OUTPUT
    ZAxisMotor : BOOL;
    EngravingMotor : BOOL;
END_VAR

VAR
    CalculatedDepth : REAL;
    CalculatedSpeed : REAL;
END_VAR

CASE DesignSelection OF
    1:
        CalculatedSpeed := 10.0;
        CalculatedDepth := 0.1;
        ZAxisMotor := TRUE;
        EngravingMotor := TRUE;
    2:
        CalculatedSpeed := 8.0;
        CalculatedDepth := 0.2;
        ZAxisMotor := TRUE;
        EngravingMotor := TRUE;
    3:
        CalculatedSpeed := 12.0;
        CalculatedDepth := 0.15;
        ZAxisMotor := TRUE;
        EngravingMotor := TRUE;
ELSE
        CalculatedSpeed := 0.0;
        CalculatedDepth := 0.0;
        ZAxisMotor := FALSE;
        EngravingMotor := FALSE;
END_CASE;

EngravingSpeed := CalculatedSpeed;
EngravingDepth := CalculatedDepth;

END_FUNCTION_BLOCK

(* ---- med_47.st ---- *)
FUNCTION_BLOCK WindowCleaningSystem
VAR_INPUT
    StartButton : BOOL;
    EmergencyStop : BOOL;
    UpperLimit : BOOL;
    LowerLimit : BOOL;
END_VAR

VAR_OUTPUT
    ElevatorUp : BOOL;
    ElevatorDown : BOOL;
    RotateClockwise : BOOL;
    WaterPump : BOOL;
    SystemFault : BOOL;
END_VAR

VAR
    CleaningInProgress : BOOL;
    CurrentState : INT; // 0=IDLE, 1=ASCENDING, 2=CLEANING_DESCENDING
    AscendTimer : TON;
    DescendTimer : TON;
    StartButtonPrev : BOOL;
    AscendTimeout : TIME := T#30S; // Maximum allowed ascent time
    DescendTimeout : TIME := T#60S; // Maximum allowed descent time
END_VAR

// Emergency Stop - Highest Priority Safety Override
IF EmergencyStop THEN
    CleaningInProgress := FALSE;
    ElevatorUp := FALSE;
    ElevatorDown := FALSE;
    RotateClockwise := FALSE;
    WaterPump := FALSE;
    CurrentState := 0;
    AscendTimer(IN:=FALSE);
    DescendTimer(IN:=FALSE);
    SystemFault := FALSE;
    RETURN; // Exit function block immediately
END_IF;

// Detect rising edge of StartButton
IF StartButton AND NOT StartButtonPrev AND NOT CleaningInProgress THEN
    CleaningInProgress := TRUE;
    CurrentState := 1; // ASCENDING state
    AscendTimer(IN:=TRUE, PT:=AscendTimeout);
    DescendTimer(IN:=FALSE);
END_IF;
StartButtonPrev := StartButton;

// Main State Machine
IF CleaningInProgress THEN
    CASE CurrentState OF
        1: // ASCENDING state
            // Safety interlock: Ensure only one direction is active
            ElevatorUp := NOT UpperLimit AND NOT LowerLimit;
            ElevatorDown := FALSE;
            RotateClockwise := FALSE;
            WaterPump := FALSE;

            // Check for upper limit or timeout
            IF UpperLimit THEN
                CurrentState := 2; // Transition to CLEANING_DESCENDING
                AscendTimer(IN:=FALSE);
                DescendTimer(IN:=TRUE, PT:=DescendTimeout);
            ELSIF AscendTimer.Q THEN
                // Timeout detected - safety fault
                CleaningInProgress := FALSE;
                CurrentState := 0;
                SystemFault := TRUE;
                ElevatorUp := FALSE;
            END_IF;

        2: // CLEANING_DESCENDING state
            // Safety interlock: Ensure only one direction is active
            ElevatorUp := FALSE;
            ElevatorDown := NOT LowerLimit AND NOT UpperLimit;
            RotateClockwise := TRUE; // Brush activates during descent
            WaterPump := TRUE;       // Pump activates during descent

            // Check for lower limit or timeout
            IF LowerLimit THEN
                CleaningInProgress := FALSE;
                CurrentState := 0; // Return to IDLE
                DescendTimer(IN:=FALSE);
                ElevatorDown := FALSE;
                RotateClockwise := FALSE;
                WaterPump := FALSE;
            ELSIF DescendTimer.Q THEN
                // Timeout detected - safety fault
                CleaningInProgress := FALSE;
                CurrentState := 0;
                SystemFault := TRUE;
                ElevatorDown := FALSE;
                RotateClockwise := FALSE;
                WaterPump := FALSE;
            END_IF;
    END_CASE;
ELSE
    // IDLE state - ensure all outputs are off
    ElevatorUp := FALSE;
    ElevatorDown := FALSE;
    RotateClockwise := FALSE;
    WaterPump := FALSE;
    CurrentState := 0;
    AscendTimer(IN:=FALSE);
    DescendTimer(IN:=FALSE);

    // Auto-reset fault if system is manually restarted
    IF StartButton AND NOT StartButtonPrev THEN
        SystemFault := FALSE;
    END_IF;
END_IF;

// Final safety interlock to prevent simultaneous up/down movement
// This is a redundant safety check
IF ElevatorUp AND ElevatorDown THEN
    ElevatorUp := FALSE;
    ElevatorDown := FALSE;
    SystemFault := TRUE;
END_IF;

END_FUNCTION_BLOCK

(* ---- med_48.st ---- *)
FUNCTION_BLOCK ChargingStationControl
VAR_INPUT
    EVConnected : BOOL;
    EVVoltage : REAL;
    EVCurrent : REAL;
    EVStateOfCharge : REAL;
    ChargingTimer : TIME;
    MinimumVoltage : REAL;
    MaximumCurrent : REAL;
    MinimumSOC : REAL;
    ChargingVoltage : REAL;
    ChargingCurrent : REAL;
    MaximumChargingTime : TIME;
END_VAR

VAR_OUTPUT
    EVCharging : BOOL;
END_VAR

VAR
    bStartConditionsMet : BOOL;
    bStopConditionsMet : BOOL;
END_VAR

(* Evaluate start conditions - ALL must be TRUE to start charging *)
bStartConditionsMet := EVConnected
    AND (EVVoltage > MinimumVoltage)
    AND (EVCurrent <= MaximumCurrent)
    AND (EVStateOfCharge < 100.0)
    AND (ChargingTimer <= MaximumChargingTime);

(* Evaluate stop conditions - ANY condition being TRUE stops charging *)
bStopConditionsMet := (NOT EVConnected)
    OR (EVVoltage <= MinimumVoltage)
    OR (EVCurrent > MaximumCurrent)
    OR (EVStateOfCharge >= 100.0)
    OR (ChargingTimer > MaximumChargingTime);

(* Main control logic *)
IF bStartConditionsMet AND NOT bStopConditionsMet THEN
    EVCharging := TRUE;
ELSE
    EVCharging := FALSE;
END_IF;

END_FUNCTION_BLOCK
